LIN {X 0,Y 153.552,Z 569.709,A -85,B 0,C 180,E1 -25423.871,E2 -25423.871} C_VEL
LIN {X 0,Y 146.34,Z 578.875,A -85,B 0,C 180,E1 -25427.749,E2 -25427.749} C_VEL
LIN {X 0,Y 140.763,Z 585.487,A -85,B 0,C 180,E1 -25431.382,E2 -25431.382} C_VEL
LIN {X 0,Y 134.19,Z 592.793,A -85,B 0,C 180,E1 -25436.638,E2 -25436.638} C_VEL
LIN {X 0,Y 128.826,Z 598.573,A -85,B 0,C 180,E1 -25442.371,E2 -25442.371} C_VEL
LIN {X 0,Y 125.476,Z 601.997,A -85,B 0,C 180,E1 -25446.915,E2 -25446.915} C_VEL
LIN {X 0,Y 122.311,Z 605.447,A -85,B 0,C 180,E1 -25453.302,E2 -25453.302} C_VEL
LIN {X 0,Y 120.389,Z 607.718,A -85,B 0,C 180,E1 -25459.912,E2 -25459.912} C_VEL
LIN {X 0,Y 119.599,Z 608.867,A -85,B 0,C 180,E1 -25466.63,E2 -25466.63} C_VEL
LIN {X 0,Y 119.528,Z 608.954,A -85,B 0,C 180,E1 -25471.681,E2 -25471.681} C_VEL
LIN {X 0,Y 119.898,Z 608.461,A -85,B 0,C 180,E1 -25476.731,E2 -25476.731} C_VEL
LIN {X 0,Y 121.179,Z 606.8,A -85,B 0,C 180,E1 -25483.413,E2 -25483.413} C_VEL
LIN {X 0,Y 123.696,Z 603.988,A -85,B 0,C 180,E1 -25489.93,E2 -25489.93} C_VEL
LIN {X 0,Y 127.583,Z 599.947,A -85,B 0,C 180,E1 -25496.146,E2 -25496.146} C_VEL
LIN {X 0,Y 132.603,Z 594.585,A -85,B 0,C 180,E1 -25502.004,E2 -25502.004} C_VEL
LIN {X 0,Y 138.944,Z 587.736,A -85,B 0,C 180,E1 -25507.37,E2 -25507.37} C_VEL
LIN {X 0,Y 146.247,Z 579.18,A -85,B 0,C 180,E1 -25512.28,E2 -25512.28} C_VEL
LIN {X 0,Y 153.435,Z 570.072,A -85,B 0,C 180,E1 -25516.17,E2 -25516.17} C_VEL
LIN {X 0,Y 159.977,Z 560.798,A -85,B 0,C 180,E1 -25519.27,E2 -25519.27} C_VEL
LIN {X 0,Y 167.681,Z 548.768,A -85,B 0,C 180,E1 -25522.287,E2 -25522.287} C_VEL
LIN {X 0,Y 174.467,Z 536.481,A -85,B 0,C 180,E1 -25524.657,E2 -25524.657} C_VEL
LIN {X 0,Y 180.497,Z 523.657,A -85,B 0,C 180,E1 -25526.588,E2 -25526.588} C_VEL
LIN {X 0,Y 185.677,Z 510.287,A -85,B 0,C 180,E1 -25528.183,E2 -25528.183} C_VEL
LIN {X 0,Y 190.275,Z 495.944,A -85,B 0,C 180,E1 -25529.435,E2 -25529.435} C_VEL
LIN {X 0,Y 194.075,Z 480.371,A -85,B 0,C 180,E1 -25530.435,E2 -25530.435} C_VEL
LIN {X 0,Y 196.56,Z 465.55,A -85,B 0,C 180,E1 -25531.094,E2 -25531.094} C_VEL
LIN {X 0,Y 199.678,Z 433.456,A -85,B 0,C 180,E1 -25531.975,E2 -25531.975} C_VEL
LIN {X 0,Y 201.434,Z 413.367,A -85,B 0,C 180,E1 -25532.537,E2 -25532.537} C_VEL
LIN {X 0,Y 196.703,Z 403.519,A -85,B 0,C 180,E1 -25536.219,E2 -25536.219} C_VEL
LIN {X 0,Y 193.073,Z 396.884,A -85,B 0,C 180,E1 -25539.518,E2 -25539.518} C_VEL
LIN {X 0,Y 190.075,Z 391.565,A -85,B 0,C 180,E1 -25542.794,E2 -25542.794} C_VEL
LIN {X 0,Y 187.731,Z 387.7,A -85,B 0,C 180,E1 -25545.916,E2 -25545.916} C_VEL
LIN {X 0,Y 185.703,Z 383.97,A -85,B 0,C 180,E1 -25549.506,E2 -25549.506} C_VEL
LIN {X 0,Y 183.861,Z 381,A -85,B 0,C 180,E1 -25554.558,E2 -25554.558} C_VEL
LIN {X 0,Y 183.557,Z 379.432,A -85,B 0,C 180,E1 -25556.707,E2 -25556.707} C_VEL
LIN {X 0,Y 183.337,Z 379.121,A -85,B 0,C 180,E1 -25560,E2 -25560} C_VEL
LIN {X 0,Y 183.568,Z 379.555,A -85,B 0,C 180,E1 -25562.949,E2 -25562.949} C_VEL
LIN {X 0,Y 185.21,Z 383.47,A -85,B 0,C 180,E1 -25569.005,E2 -25569.005} C_VEL
LIN {X 0,Y 185.94,Z 384.419,A -85,B 0,C 180,E1 -25570.491,E2 -25570.491} C_VEL
LIN {X 0,Y 188.426,Z 388.76,A -85,B 0,C 180,E1 -25574.582,E2 -25574.582} C_VEL
LIN {X 0,Y 190.981,Z 393.14,A -85,B 0,C 180,E1 -25577.773,E2 -25577.773} C_VEL
LIN {X 0,Y 193.616,Z 397.814,A -85,B 0,C 180,E1 -25580.518,E2 -25580.518} C_VEL
LIN {X 0,Y 196.945,Z 405.983,A -85,B 0,C 180,E1 -25583.669,E2 -25583.669} C_VEL
LIN {X 0,Y 200.304,Z 415.239,A -85,B 0,C 180,E1 -25586.483,E2 -25586.483} C_VEL
LIN {X 0,Y 201.157,Z 417.755,A -85,B 0,C 180,E1 -25587.153,E2 -25587.153} C_VEL
LIN {X 0,Y 196.088,Z 472.023,A -85,B 0,C 180,E1 -25588.616,E2 -25588.616} C_VEL
LIN {X 0,Y 193.318,Z 487.832,A -85,B 0,C 180,E1 -25589.25,E2 -25589.25} C_VEL
LIN {X 0,Y 189.505,Z 503.063,A -85,B 0,C 180,E1 -25590.168,E2 -25590.168} C_VEL
LIN {X 0,Y 184.942,Z 516.79,A -85,B 0,C 180,E1 -25591.239,E2 -25591.239} C_VEL
LIN {X 0,Y 179.479,Z 530.244,A -85,B 0,C 180,E1 -25592.661,E2 -25592.661} C_VEL
LIN {X 0,Y 173.308,Z 543.167,A -85,B 0,C 180,E1 -25594.487,E2 -25594.487} C_VEL
LIN {X 0,Y 166.611,Z 555.308,A -85,B 0,C 180,E1 -25596.732,E2 -25596.732} C_VEL
LIN {X 0,Y 159.273,Z 566.801,A -85,B 0,C 180,E1 -25599.45,E2 -25599.45} C_VEL
LIN {X 0,Y 152.418,Z 576.486,A -85,B 0,C 180,E1 -25602.461,E2 -25602.461} C_VEL
LIN {X 0,Y 145.046,Z 586.009,A -85,B 0,C 180,E1 -25606.335,E2 -25606.335} C_VEL
LIN {X 0,Y 138.531,Z 593.959,A -85,B 0,C 180,E1 -25610.644,E2 -25610.644} C_VEL
LIN {X 0,Y 131.988,Z 601.387,A -85,B 0,C 180,E1 -25616.008,E2 -25616.008} C_VEL
LIN {X 0,Y 127.784,Z 606.137,A -85,B 0,C 180,E1 -25620.565,E2 -25620.565} C_VEL
LIN {X 0,Y 125.367,Z 608.182,A -85,B 0,C 180,E1 -25622.835,E2 -25622.835} C_VEL
LIN {X 0,Y 120.068,Z 611.099,A -85,B 0,C 180,E1 -25626.514,E2 -25626.514} C_VEL
LIN {X 0,Y 116.037,Z 613.032,A -85,B 0,C 180,E1 -25629.711,E2 -25629.711} C_VEL
LIN {X 0,Y 113.983,Z 614.267,A -85,B 0,C 180,E1 -25632.41,E2 -25632.41} C_VEL
LIN {X 0,Y 113.609,Z 614.613,A -85,B 0,C 180,E1 -25633.367,E2 -25633.367} C_VEL
LIN {X 0,Y 112.455,Z 616.484,A -85,B 0,C 180,E1 -25639.195,E2 -25639.195} C_VEL
LIN {X 0,Y 112.168,Z 617.688,A -85,B 0,C 180,E1 -25646.409,E2 -25646.409} C_VEL
LIN {X 0,Y 112.361,Z 617.854,A -85,B 0,C 180,E1 -25650.002,E2 -25650.002} C_VEL
LIN {X 0,Y 112.191,Z 617.211,A -85,B 0,C 180,E1 -25657.199,E2 -25657.199} C_VEL
LIN {X 0,Y 113.057,Z 615.402,A -85,B 0,C 180,E1 -25664.4,E2 -25664.4} C_VEL
LIN {X 0,Y 115.446,Z 612.422,A -85,B 0,C 180,E1 -25671.426,E2 -25671.426} C_VEL
LIN {X 0,Y 119.303,Z 608.201,A -85,B 0,C 180,E1 -25678.119,E2 -25678.119} C_VEL
LIN {X 0,Y 124.542,Z 602.629,A -85,B 0,C 180,E1 -25684.356,E2 -25684.356} C_VEL
LIN {X 0,Y 131.241,Z 595.569,A -85,B 0,C 180,E1 -25689.988,E2 -25689.988} C_VEL
LIN {X 0,Y 137.341,Z 588.55,A -85,B 0,C 180,E1 -25694.242,E2 -25694.242} C_VEL
LIN {X 0,Y 145.382,Z 578.944,A -85,B 0,C 180,E1 -25698.531,E2 -25698.531} C_VEL
LIN {X 0,Y 153.568,Z 568.039,A -85,B 0,C 180,E1 -25702.135,E2 -25702.135} C_VEL
LIN {X 0,Y 161.782,Z 555.793,A -85,B 0,C 180,E1 -25705.082,E2 -25705.082} C_VEL
LIN {X 0,Y 168.964,Z 543.304,A -85,B 0,C 180,E1 -25707.385,E2 -25707.385} C_VEL
LIN {X 0,Y 175.041,Z 531.032,A -85,B 0,C 180,E1 -25709.119,E2 -25709.119} C_VEL
LIN {X 0,Y 180.613,Z 517.76,A -85,B 0,C 180,E1 -25710.537,E2 -25710.537} C_VEL
LIN {X 0,Y 185.274,Z 504.367,A -85,B 0,C 180,E1 -25711.593,E2 -25711.593} C_VEL
LIN {X 0,Y 189.234,Z 489.693,A -85,B 0,C 180,E1 -25712.464,E2 -25712.464} C_VEL
LIN {X 0,Y 192.151,Z 474.204,A -85,B 0,C 180,E1 -25713.128,E2 -25713.128} C_VEL
LIN {X 0,Y 194.293,Z 455.279,A -85,B 0,C 180,E1 -25713.639,E2 -25713.639} C_VEL
LIN {X 0,Y 197.478,Z 420.453,A -85,B 0,C 180,E1 -25714.578,E2 -25714.578} C_VEL
LIN {X 0,Y 194.285,Z 411.099,A -85,B 0,C 180,E1 -25717.467,E2 -25717.467} C_VEL
LIN {X 0,Y 191.368,Z 403.557,A -85,B 0,C 180,E1 -25720.442,E2 -25720.442} C_VEL
LIN {X 0,Y 188.462,Z 398.084,A -85,B 0,C 180,E1 -25723.759,E2 -25723.759} C_VEL
LIN {X 0,Y 186.121,Z 394.028,A -85,B 0,C 180,E1 -25727.044,E2 -25727.044} C_VEL
LIN {X 0,Y 184.324,Z 390.657,A -85,B 0,C 180,E1 -25730.398,E2 -25730.398} C_VEL
LIN {X 0,Y 182.51,Z 387.017,A -85,B 0,C 180,E1 -25736.136,E2 -25736.136} C_VEL
LIN {X 0,Y 182.38,Z 386.274,A -85,B 0,C 180,E1 -25737.239,E2 -25737.239} C_VEL
LIN {X 0,Y 182.237,Z 386.167,A -85,B 0,C 180,E1 -25742.21,E2 -25742.21} C_VEL
LIN {X 0,Y 182.454,Z 386.689,A -85,B 0,C 180,E1 -25744.004,E2 -25744.004} C_VEL
LIN {X 0,Y 183.802,Z 390.149,A -85,B 0,C 180,E1 -25749.075,E2 -25749.075} C_VEL
LIN {X 0,Y 184.618,Z 391.329,A -85,B 0,C 180,E1 -25750.834,E2 -25750.834} C_VEL
LIN {X 0,Y 186.972,Z 395.589,A -85,B 0,C 180,E1 -25754.837,E2 -25754.837} C_VEL
LIN {X 0,Y 189.331,Z 399.838,A -85,B 0,C 180,E1 -25757.904,E2 -25757.904} C_VEL
LIN {X 0,Y 192.068,Z 404.893,A -85,B 0,C 180,E1 -25760.849,E2 -25760.849} C_VEL
LIN {X 0,Y 195.488,Z 411.77,A -85,B 0,C 180,E1 -25763.998,E2 -25763.998} C_VEL
LIN {X 0,Y 197.747,Z 416.775,A -85,B 0,C 180,E1 -25765.862,E2 -25765.862} C_VEL
LIN {X 0,Y 193.157,Z 465.028,A -85,B 0,C 180,E1 -25767.189,E2 -25767.189} C_VEL
LIN {X 0,Y 190.472,Z 480.44,A -85,B 0,C 180,E1 -25767.82,E2 -25767.82} C_VEL
LIN {X 0,Y 186.85,Z 495.126,A -85,B 0,C 180,E1 -25768.732,E2 -25768.732} C_VEL
LIN {X 0,Y 182.161,Z 509.686,A -85,B 0,C 180,E1 -25769.984,E2 -25769.984} C_VEL
LIN {X 0,Y 177.053,Z 522.601,A -85,B 0,C 180,E1 -25771.474,E2 -25771.474} C_VEL
LIN {X 0,Y 170.555,Z 536.147,A -85,B 0,C 180,E1 -25773.441,E2 -25773.441} C_VEL
LIN {X 0,Y 163.521,Z 548.533,A -85,B 0,C 180,E1 -25775.781,E2 -25775.781} C_VEL
LIN {X 0,Y 156.694,Z 558.904,A -85,B 0,C 180,E1 -25778.286,E2 -25778.286} C_VEL
LIN {X 0,Y 149.799,Z 568.511,A -85,B 0,C 180,E1 -25781.35,E2 -25781.35} C_VEL
LIN {X 0,Y 143.255,Z 576.708,A -85,B 0,C 180,E1 -25784.652,E2 -25784.652} C_VEL
LIN {X 0,Y 136.203,Z 584.763,A -85,B 0,C 180,E1 -25788.858,E2 -25788.858} C_VEL
LIN {X 0,Y 129.928,Z 591.404,A -85,B 0,C 180,E1 -25793.485,E2 -25793.485} C_VEL
LIN {X 0,Y 123.831,Z 597.54,A -85,B 0,C 180,E1 -25799.281,E2 -25799.281} C_VEL
LIN {X 0,Y 118.956,Z 602.269,A -85,B 0,C 180,E1 -25805.569,E2 -25805.569} C_VEL
LIN {X 0,Y 115.513,Z 605.719,A -85,B 0,C 180,E1 -25812.288,E2 -25812.288} C_VEL
LIN {X 0,Y 113.386,Z 607.989,A -85,B 0,C 180,E1 -25819.282,E2 -25819.282} C_VEL
LIN {X 0,Y 112.523,Z 609.137,A -85,B 0,C 180,E1 -25826.417,E2 -25826.417} C_VEL
LIN {X 0,Y 112.46,Z 609.266,A -85,B 0,C 180,E1 -25830.803,E2 -25830.803} C_VEL
LIN {X 0,Y 112.854,Z 608.731,A -85,B 0,C 180,E1 -25837.153,E2 -25837.153} C_VEL
LIN {X 0,Y 114.26,Z 607.071,A -85,B 0,C 180,E1 -25844.241,E2 -25844.241} C_VEL
LIN {X 0,Y 117.025,Z 604.258,A -85,B 0,C 180,E1 -25851.119,E2 -25851.119} C_VEL
LIN {X 0,Y 121.225,Z 600.217,A -85,B 0,C 180,E1 -25857.631,E2 -25857.631} C_VEL
LIN {X 0,Y 126.622,Z 594.855,A -85,B 0,C 180,E1 -25863.712,E2 -25863.712} C_VEL
LIN {X 0,Y 133.356,Z 588.005,A -85,B 0,C 180,E1 -25869.227,E2 -25869.227} C_VEL
LIN {X 0,Y 141.056,Z 579.449,A -85,B 0,C 180,E1 -25874.228,E2 -25874.228} C_VEL
LIN {X 0,Y 147.522,Z 571.748,A -85,B 0,C 180,E1 -25877.596,E2 -25877.596} C_VEL
LIN {X 0,Y 154.236,Z 562.683,A -85,B 0,C 180,E1 -25880.77,E2 -25880.77} C_VEL
LIN {X 0,Y 161.56,Z 551.969,A -85,B 0,C 180,E1 -25883.586,E2 -25883.586} C_VEL
LIN {X 0,Y 168.484,Z 540.271,A -85,B 0,C 180,E1 -25886,E2 -25886} C_VEL
LIN {X 0,Y 174.929,Z 527.738,A -85,B 0,C 180,E1 -25887.974,E2 -25887.974} C_VEL
LIN {X 0,Y 180.224,Z 515.305,A -85,B 0,C 180,E1 -25889.573,E2 -25889.573} C_VEL
LIN {X 0,Y 185.061,Z 501.838,A -85,B 0,C 180,E1 -25890.862,E2 -25890.862} C_VEL
LIN {X 0,Y 189.202,Z 487.184,A -85,B 0,C 180,E1 -25891.908,E2 -25891.908} C_VEL
LIN {X 0,Y 192.295,Z 471.921,A -85,B 0,C 180,E1 -25892.71,E2 -25892.71} C_VEL
LIN {X 0,Y 194.29,Z 456.851,A -85,B 0,C 180,E1 -25893.198,E2 -25893.198} C_VEL
LIN {X 0,Y 198,Z 416.982,A -85,B 0,C 180,E1 -25894.238,E2 -25894.238} C_VEL
LIN {X 0,Y 194.142,Z 408.687,A -85,B 0,C 180,E1 -25897.519,E2 -25897.519} C_VEL
LIN {X 0,Y 190.419,Z 401.503,A -85,B 0,C 180,E1 -25901.263,E2 -25901.263} C_VEL
LIN {X 0,Y 188.03,Z 397.319,A -85,B 0,C 180,E1 -25904.152,E2 -25904.152} C_VEL
LIN {X 0,Y 186.393,Z 394.382,A -85,B 0,C 180,E1 -25906.546,E2 -25906.546} C_VEL
LIN {X 0,Y 184.5,Z 390.792,A -85,B 0,C 180,E1 -25910.13,E2 -25910.13} C_VEL
LIN {X 0,Y 182.75,Z 387.32,A -85,B 0,C 180,E1 -25915.865,E2 -25915.865} C_VEL
LIN {X 0,Y 182.622,Z 386.361,A -85,B 0,C 180,E1 -25917.242,E2 -25917.242} C_VEL
LIN {X 0,Y 182.617,Z 386.338,A -85,B 0,C 180,E1 -25922.205,E2 -25922.205} C_VEL
LIN {X 0,Y 184.348,Z 390.581,A -85,B 0,C 180,E1 -25929.048,E2 -25929.048} C_VEL
LIN {X 0,Y 184.802,Z 391.299,A -85,B 0,C 180,E1 -25930.026,E2 -25930.026} C_VEL
LIN {X 0,Y 187.075,Z 395.482,A -85,B 0,C 180,E1 -25933.995,E2 -25933.995} C_VEL
LIN {X 0,Y 189.336,Z 399.547,A -85,B 0,C 180,E1 -25936.996,E2 -25936.996} C_VEL
LIN {X 0,Y 191.684,Z 403.991,A -85,B 0,C 180,E1 -25939.615,E2 -25939.615} C_VEL
LIN {X 0,Y 194.459,Z 411.21,A -85,B 0,C 180,E1 -25942.455,E2 -25942.455} C_VEL
LIN {X 0,Y 197.488,Z 420.003,A -85,B 0,C 180,E1 -25945.209,E2 -25945.209} C_VEL
LIN {X 0,Y 197.736,Z 420.842,A -85,B 0,C 180,E1 -25945.429,E2 -25945.429} C_VEL
LIN {X 0,Y 192.751,Z 471.989,A -85,B 0,C 180,E1 -25946.769,E2 -25946.769} C_VEL
LIN {X 0,Y 189.948,Z 487.57,A -85,B 0,C 180,E1 -25947.38,E2 -25947.38} C_VEL
LIN {X 0,Y 186.032,Z 502.8,A -85,B 0,C 180,E1 -25948.274,E2 -25948.274} C_VEL
LIN {X 0,Y 181.359,Z 516.525,A -85,B 0,C 180,E1 -25949.32,E2 -25949.32} C_VEL
LIN {X 0,Y 175.741,Z 529.978,A -85,B 0,C 180,E1 -25950.708,E2 -25950.708} C_VEL
LIN {X 0,Y 168.962,Z 543.687,A -85,B 0,C 180,E1 -25952.618,E2 -25952.618} C_VEL
LIN {X 0,Y 161.8,Z 556.113,A -85,B 0,C 180,E1 -25954.931,E2 -25954.931} C_VEL
LIN {X 0,Y 153.607,Z 568.295,A -85,B 0,C 180,E1 -25957.887,E2 -25957.887} C_VEL
LIN {X 0,Y 145.38,Z 579.146,A -85,B 0,C 180,E1 -25961.472,E2 -25961.472} C_VEL
LIN {X 0,Y 137.695,Z 588.394,A -85,B 0,C 180,E1 -25965.607,E2 -25965.607} C_VEL
LIN {X 0,Y 131.243,Z 595.726,A -85,B 0,C 180,E1 -25970.016,E2 -25970.016} C_VEL
LIN {X 0,Y 124.559,Z 602.748,A -85,B 0,C 180,E1 -25975.653,E2 -25975.653} C_VEL
LIN {X 0,Y 118.779,Z 608.82,A -85,B 0,C 180,E1 -25982.564,E2 -25982.564} C_VEL
LIN {X 0,Y 115.444,Z 612.489,A -85,B 0,C 180,E1 -25988.578,E2 -25988.578} C_VEL
LIN {X 0,Y 113.609,Z 614.613,A -85,B 0,C 180,E1 -25993.367,E2 -25993.367} C_VEL
LIN {X 0,Y 112.237,Z 615.668,A -85,B 0,C 180,E1 -25996.238,E2 -25996.238} C_VEL
LIN {X 0,Y 108.69,Z 616.831,A -85,B 0,C 180,E1 -26001.006,E2 -26001.006} C_VEL
LIN {X 0,Y 106.114,Z 617.35,A -85,B 0,C 180,E1 -26005.038,E2 -26005.038} C_VEL
LIN {X 0,Y 105.198,Z 617.515,A -85,B 0,C 180,E1 -26008.232,E2 -26008.232} C_VEL
LIN {X 0,Y 105.202,Z 617.554,A -85,B 0,C 180,E1 -26009.314,E2 -26009.314} C_VEL
LIN {X 0,Y 105.081,Z 617.411,A -85,B 0,C 180,E1 -26013.837,E2 -26013.837} C_VEL
LIN {X 0,Y 105.455,Z 616.179,A -85,B 0,C 180,E1 -26021.535,E2 -26021.535} C_VEL
LIN {X 0,Y 107.235,Z 613.787,A -85,B 0,C 180,E1 -26029.131,E2 -26029.131} C_VEL
LIN {X 0,Y 110.722,Z 610.198,A -85,B 0,C 180,E1 -26036.382,E2 -26036.382} C_VEL
LIN {X 0,Y 115.67,Z 605.317,A -85,B 0,C 180,E1 -26043.152,E2 -26043.152} C_VEL
LIN {X 0,Y 122.065,Z 599.021,A -85,B 0,C 180,E1 -26049.299,E2 -26049.299} C_VEL
LIN {X 0,Y 128.724,Z 592.235,A -85,B 0,C 180,E1 -26054.118,E2 -26054.118} C_VEL
LIN {X 0,Y 136.134,Z 584.034,A -85,B 0,C 180,E1 -26058.469,E2 -26058.469} C_VEL
LIN {X 0,Y 144.342,Z 574.22,A -85,B 0,C 180,E1 -26062.301,E2 -26062.301} C_VEL
LIN {X 0,Y 151.875,Z 564.194,A -85,B 0,C 180,E1 -26065.226,E2 -26065.226} C_VEL
LIN {X 0,Y 159.467,Z 552.848,A -85,B 0,C 180,E1 -26067.734,E2 -26067.734} C_VEL
LIN {X 0,Y 166.593,Z 540.433,A -85,B 0,C 180,E1 -26069.865,E2 -26069.865} C_VEL
LIN {X 0,Y 172.931,Z 527.625,A -85,B 0,C 180,E1 -26071.507,E2 -26071.507} C_VEL
LIN {X 0,Y 178.678,Z 513.643,A -85,B 0,C 180,E1 -26072.865,E2 -26072.865} C_VEL
LIN {X 0,Y 183.496,Z 499.24,A -85,B 0,C 180,E1 -26073.856,E2 -26073.856} C_VEL
LIN {X 0,Y 187.171,Z 484.445,A -85,B 0,C 180,E1 -26074.63,E2 -26074.63} C_VEL
LIN {X 0,Y 189.572,Z 470.621,A -85,B 0,C 180,E1 -26075.143,E2 -26075.143} C_VEL
LIN {X 0,Y 194.235,Z 423.709,A -85,B 0,C 180,E1 -26076.35,E2 -26076.35} C_VEL
LIN {X 0,Y 191.745,Z 415.955,A -85,B 0,C 180,E1 -26078.851,E2 -26078.851} C_VEL
LIN {X 0,Y 189.449,Z 409.614,A -85,B 0,C 180,E1 -26081.41,E2 -26081.41} C_VEL
LIN {X 0,Y 186.753,Z 404.322,A -85,B 0,C 180,E1 -26084.727,E2 -26084.727} C_VEL
LIN {X 0,Y 184.823,Z 400.755,A -85,B 0,C 180,E1 -26087.65,E2 -26087.65} C_VEL
LIN {X 0,Y 183.263,Z 397.581,A -85,B 0,C 180,E1 -26090.759,E2 -26090.759} C_VEL
LIN {X 0,Y 181.61,Z 394.108,A -85,B 0,C 180,E1 -26096.256,E2 -26096.256} C_VEL
LIN {X 0,Y 181.442,Z 393.23,A -85,B 0,C 180,E1 -26097.78,E2 -26097.78} C_VEL
LIN {X 0,Y 181.43,Z 393.295,A -85,B 0,C 180,E1 -26102.776,E2 -26102.776} C_VEL
LIN {X 0,Y 181.639,Z 394.346,A -85,B 0,C 180,E1 -26104.577,E2 -26104.577} C_VEL
LIN {X 0,Y 183.057,Z 397.424,A -85,B 0,C 180,E1 -26109.391,E2 -26109.391} C_VEL
LIN {X 0,Y 183.734,Z 398.826,A -85,B 0,C 180,E1 -26110.922,E2 -26110.922} C_VEL
LIN {X 0,Y 185.722,Z 402.449,A -85,B 0,C 180,E1 -26114.379,E2 -26114.379} C_VEL
LIN {X 0,Y 188.542,Z 407.745,A -85,B 0,C 180,E1 -26118.122,E2 -26118.122} C_VEL
LIN {X 0,Y 191.93,Z 414.739,A -85,B 0,C 180,E1 -26121.748,E2 -26121.748} C_VEL
LIN {X 0,Y 194.481,Z 420.422,A -85,B 0,C 180,E1 -26124.101,E2 -26124.101} C_VEL
LIN {X 0,Y 190.029,Z 465.302,A -85,B 0,C 180,E1 -26125.291,E2 -26125.291} C_VEL
LIN {X 0,Y 187.451,Z 479.864,A -85,B 0,C 180,E1 -26125.863,E2 -26125.863} C_VEL
LIN {X 0,Y 183.541,Z 495.404,A -85,B 0,C 180,E1 -26126.788,E2 -26126.788} C_VEL
LIN {X 0,Y 178.728,Z 509.962,A -85,B 0,C 180,E1 -26128.017,E2 -26128.017} C_VEL
LIN {X 0,Y 173.336,Z 523.154,A -85,B 0,C 180,E1 -26129.51,E2 -26129.51} C_VEL
LIN {X 0,Y 166.76,Z 536.421,A -85,B 0,C 180,E1 -26131.411,E2 -26131.411} C_VEL
LIN {X 0,Y 159.474,Z 548.807,A -85,B 0,C 180,E1 -26133.712,E2 -26133.712} C_VEL
LIN {X 0,Y 152.396,Z 559.178,A -85,B 0,C 180,E1 -26136.189,E2 -26136.189} C_VEL
LIN {X 0,Y 145.179,Z 568.785,A -85,B 0,C 180,E1 -26139.234,E2 -26139.234} C_VEL
LIN {X 0,Y 138.352,Z 576.981,A -85,B 0,C 180,E1 -26142.558,E2 -26142.558} C_VEL
LIN {X 0,Y 130.922,Z 585.036,A -85,B 0,C 180,E1 -26146.807,E2 -26146.807} C_VEL
LIN {X 0,Y 124.262,Z 591.678,A -85,B 0,C 180,E1 -26151.525,E2 -26151.525} C_VEL
LIN {X 0,Y 117.751,Z 597.814,A -85,B 0,C 180,E1 -26157.507,E2 -26157.507} C_VEL
LIN {X 0,Y 112.515,Z 602.541,A -85,B 0,C 180,E1 -26164.07,E2 -26164.07} C_VEL
LIN {X 0,Y 108.762,Z 605.99,A -85,B 0,C 180,E1 -26171.148,E2 -26171.148} C_VEL
LIN {X 0,Y 106.409,Z 608.261,A -85,B 0,C 180,E1 -26178.57,E2 -26178.57} C_VEL
LIN {X 0,Y 105.455,Z 609.407,A -85,B 0,C 180,E1 -26186.177,E2 -26186.177} C_VEL
LIN {X 0,Y 105.392,Z 609.558,A -85,B 0,C 180,E1 -26189.998,E2 -26189.998} C_VEL
LIN {X 0,Y 105.807,Z 609.001,A -85,B 0,C 180,E1 -26197.632,E2 -26197.632} C_VEL
LIN {X 0,Y 107.38,Z 607.342,A -85,B 0,C 180,E1 -26205.175,E2 -26205.175} C_VEL
LIN {X 0,Y 110.393,Z 604.529,A -85,B 0,C 180,E1 -26212.455,E2 -26212.455} C_VEL
LIN {X 0,Y 114.961,Z 600.488,A -85,B 0,C 180,E1 -26219.278,E2 -26219.278} C_VEL
LIN {X 0,Y 120.749,Z 595.126,A -85,B 0,C 180,E1 -26225.592,E2 -26225.592} C_VEL
LIN {X 0,Y 127.898,Z 588.276,A -85,B 0,C 180,E1 -26231.252,E2 -26231.252} C_VEL
LIN {X 0,Y 136.043,Z 579.719,A -85,B 0,C 180,E1 -26236.321,E2 -26236.321} C_VEL
LIN {X 0,Y 142.807,Z 572.017,A -85,B 0,C 180,E1 -26239.71,E2 -26239.71} C_VEL
LIN {X 0,Y 149.839,Z 562.951,A -85,B 0,C 180,E1 -26242.877,E2 -26242.877} C_VEL
LIN {X 0,Y 157.449,Z 552.236,A -85,B 0,C 180,E1 -26245.665,E2 -26245.665} C_VEL
LIN {X 0,Y 164.623,Z 540.537,A -85,B 0,C 180,E1 -26248.046,E2 -26248.046} C_VEL
LIN {X 0,Y 171.771,Z 526.96,A -85,B 0,C 180,E1 -26250.13,E2 -26250.13} C_VEL
LIN {X 0,Y 177.492,Z 513.632,A -85,B 0,C 180,E1 -26251.763,E2 -26251.763} C_VEL
LIN {X 0,Y 182.758,Z 498.723,A -85,B 0,C 180,E1 -26253.083,E2 -26253.083} C_VEL
LIN {X 0,Y 186.857,Z 483.643,A -85,B 0,C 180,E1 -26254.045,E2 -26254.045} C_VEL
LIN {X 0,Y 189.664,Z 468.983,A -85,B 0,C 180,E1 -26254.725,E2 -26254.725} C_VEL
LIN {X 0,Y 191.551,Z 453.831,A -85,B 0,C 180,E1 -26255.153,E2 -26255.153} C_VEL
LIN {X 0,Y 194.707,Z 420.604,A -85,B 0,C 180,E1 -26256.023,E2 -26256.023} C_VEL
LIN {X 0,Y 191.485,Z 413.416,A -85,B 0,C 180,E1 -26259.056,E2 -26259.056} C_VEL
LIN {X 0,Y 188.157,Z 406.822,A -85,B 0,C 180,E1 -26262.753,E2 -26262.753} C_VEL
LIN {X 0,Y 186.031,Z 402.882,A -85,B 0,C 180,E1 -26265.645,E2 -26265.645} C_VEL
LIN {X 0,Y 184.963,Z 400.87,A -85,B 0,C 180,E1 -26267.38,E2 -26267.38} C_VEL
LIN {X 0,Y 183.383,Z 397.654,A -85,B 0,C 180,E1 -26270.626,E2 -26270.626} C_VEL
LIN {X 0,Y 181.802,Z 394.148,A -85,B 0,C 180,E1 -26276.398,E2 -26276.398} C_VEL
LIN {X 0,Y 181.701,Z 393.312,A -85,B 0,C 180,E1 -26277.783,E2 -26277.783} C_VEL
LIN {X 0,Y 181.743,Z 393.458,A -85,B 0,C 180,E1 -26282.216,E2 -26282.216} C_VEL
LIN {X 0,Y 183.238,Z 397.453,A -85,B 0,C 180,E1 -26288.547,E2 -26288.547} C_VEL
LIN {X 0,Y 183.771,Z 398.434,A -85,B 0,C 180,E1 -26289.782,E2 -26289.782} C_VEL
LIN {X 0,Y 185.745,Z 402.2,A -85,B 0,C 180,E1 -26293.4,E2 -26293.4} C_VEL
LIN {X 0,Y 188.113,Z 406.656,A -85,B 0,C 180,E1 -26296.691,E2 -26296.691} C_VEL
LIN {X 0,Y 190.081,Z 410.84,A -85,B 0,C 180,E1 -26299.016,E2 -26299.016} C_VEL
LIN {X 0,Y 192.584,Z 418.01,A -85,B 0,C 180,E1 -26301.754,E2 -26301.754} C_VEL
LIN {X 0,Y 194.489,Z 423.973,A -85,B 0,C 180,E1 -26303.643,E2 -26303.643} C_VEL
LIN {X 0,Y 189.624,Z 471.934,A -85,B 0,C 180,E1 -26304.858,E2 -26304.858} C_VEL
LIN {X 0,Y 186.789,Z 487.309,A -85,B 0,C 180,E1 -26305.446,E2 -26305.446} C_VEL
LIN {X 0,Y 182.775,Z 502.536,A -85,B 0,C 180,E1 -26306.313,E2 -26306.313} C_VEL
LIN {X 0,Y 177.979,Z 516.26,A -85,B 0,C 180,E1 -26307.32,E2 -26307.32} C_VEL
LIN {X 0,Y 172.212,Z 529.711,A -85,B 0,C 180,E1 -26308.669,E2 -26308.669} C_VEL
LIN {X 0,Y 165.233,Z 543.42,A -85,B 0,C 180,E1 -26310.538,E2 -26310.538} C_VEL
LIN {X 0,Y 157.821,Z 555.845,A -85,B 0,C 180,E1 -26312.806,E2 -26312.806} C_VEL
LIN {X 0,Y 149.325,Z 568.026,A -85,B 0,C 180,E1 -26315.723,E2 -26315.723} C_VEL
LIN {X 0,Y 140.739,Z 578.875,A -85,B 0,C 180,E1 -26319.286,E2 -26319.286} C_VEL
LIN {X 0,Y 133.934,Z 586.709,A -85,B 0,C 180,E1 -26322.726,E2 -26322.726} C_VEL
LIN {X 0,Y 125.829,Z 595.454,A -85,B 0,C 180,E1 -26327.916,E2 -26327.916} C_VEL
LIN {X 0,Y 118.7,Z 602.476,A -85,B 0,C 180,E1 -26333.697,E2 -26333.697} C_VEL
LIN {X 0,Y 112.979,Z 608.014,A -85,B 0,C 180,E1 -26340.157,E2 -26340.157} C_VEL
LIN {X 0,Y 108.787,Z 612.216,A -85,B 0,C 180,E1 -26347.195,E2 -26347.195} C_VEL
LIN {X 0,Y 106.14,Z 615.176,A -85,B 0,C 180,E1 -26354.643,E2 -26354.643} C_VEL
LIN {X 0,Y 105.119,Z 616.959,A -85,B 0,C 180,E1 -26362.318,E2 -26362.318} C_VEL
LIN {X 0,Y 105.202,Z 617.554,A -85,B 0,C 180,E1 -26369.314,E2 -26369.314} C_VEL
LIN {X 0,Y 105.014,Z 617.581,A -85,B 0,C 180,E1 -26371.442,E2 -26371.442} C_VEL
LIN {X 0,Y 103.723,Z 617.402,A -85,B 0,C 180,E1 -26374.605,E2 -26374.605} C_VEL
LIN {X 0,Y 99.655,Z 616.073,A -85,B 0,C 180,E1 -26382.167,E2 -26382.167} C_VEL
LIN {X 0,Y 99.123,Z 615.13,A -85,B 0,C 180,E1 -26385.587,E2 -26385.587} C_VEL
LIN {X 0,Y 99.307,Z 614.768,A -85,B 0,C 180,E1 -26386.723,E2 -26386.723} C_VEL
LIN {X 0,Y 102.205,Z 611.873,A -85,B 0,C 180,E1 -26394.369,E2 -26394.369} C_VEL
LIN {X 0,Y 106.825,Z 607.651,A -85,B 0,C 180,E1 -26401.759,E2 -26401.759} C_VEL
LIN {X 0,Y 112.978,Z 602.08,A -85,B 0,C 180,E1 -26408.469,E2 -26408.469} C_VEL
LIN {X 0,Y 120.601,Z 595.02,A -85,B 0,C 180,E1 -26414.373,E2 -26414.373} C_VEL
LIN {X 0,Y 128.146,Z 587.334,A -85,B 0,C 180,E1 -26419.089,E2 -26419.089} C_VEL
LIN {X 0,Y 136.315,Z 578.393,A -85,B 0,C 180,E1 -26423.05,E2 -26423.05} C_VEL
LIN {X 0,Y 145.233,Z 567.49,A -85,B 0,C 180,E1 -26426.592,E2 -26426.592} C_VEL
LIN {X 0,Y 154.053,Z 555.242,A -85,B 0,C 180,E1 -26429.442,E2 -26429.442} C_VEL
LIN {X 0,Y 161.721,Z 542.752,A -85,B 0,C 180,E1 -26431.647,E2 -26431.647} C_VEL
LIN {X 0,Y 168.18,Z 530.48,A -85,B 0,C 180,E1 -26433.285,E2 -26433.285} C_VEL
LIN {X 0,Y 174.048,Z 517.206,A -85,B 0,C 180,E1 -26434.624,E2 -26434.624} C_VEL
LIN {X 0,Y 179.342,Z 502.683,A -85,B 0,C 180,E1 -26435.663,E2 -26435.663} C_VEL
LIN {X 0,Y 183.483,Z 487.607,A -85,B 0,C 180,E1 -26436.478,E2 -26436.478} C_VEL
LIN {X 0,Y 186.382,Z 472.363,A -85,B 0,C 180,E1 -26437.064,E2 -26437.064} C_VEL
LIN {X 0,Y 189.938,Z 439.628,A -85,B 0,C 180,E1 -26437.862,E2 -26437.862} C_VEL
LIN {X 0,Y 191.119,Z 426.649,A -85,B 0,C 180,E1 -26438.26,E2 -26438.26} C_VEL
LIN {X 0,Y 188.829,Z 419.293,A -85,B 0,C 180,E1 -26440.853,E2 -26440.853} C_VEL
LIN {X 0,Y 187.251,Z 414.935,A -85,B 0,C 180,E1 -26442.809,E2 -26442.809} C_VEL
LIN {X 0,Y 184.969,Z 410.31,A -85,B 0,C 180,E1 -26445.906,E2 -26445.906} C_VEL
LIN {X 0,Y 183.474,Z 407.325,A -85,B 0,C 180,E1 -26448.399,E2 -26448.399} C_VEL
LIN {X 0,Y 182.089,Z 404.363,A -85,B 0,C 180,E1 -26451.399,E2 -26451.399} C_VEL
LIN {X 0,Y 180.646,Z 400.826,A -85,B 0,C 180,E1 -26456.926,E2 -26456.926} C_VEL
LIN {X 0,Y 180.572,Z 400.32,A -85,B 0,C 180,E1 -26457.77,E2 -26457.77} C_VEL
LIN {X 0,Y 180.508,Z 400.258,A -85,B 0,C 180,E1 -26462.232,E2 -26462.232} C_VEL
LIN {X 0,Y 180.644,Z 400.903,A -85,B 0,C 180,E1 -26463.695,E2 -26463.695} C_VEL
LIN {X 0,Y 181.955,Z 404.282,A -85,B 0,C 180,E1 -26468.888,E2 -26468.888} C_VEL
LIN {X 0,Y 182.501,Z 405.472,A -85,B 0,C 180,E1 -26470.225,E2 -26470.225} C_VEL
LIN {X 0,Y 184.314,Z 409.02,A -85,B 0,C 180,E1 -26473.647,E2 -26473.647} C_VEL
LIN {X 0,Y 186.385,Z 413.192,A -85,B 0,C 180,E1 -26476.674,E2 -26476.674} C_VEL
LIN {X 0,Y 189.381,Z 419.498,A -85,B 0,C 180,E1 -26480.218,E2 -26480.218} C_VEL
LIN {X 0,Y 191.351,Z 424.086,A -85,B 0,C 180,E1 -26482.242,E2 -26482.242} C_VEL
LIN {X 0,Y 187.055,Z 465.958,A -85,B 0,C 180,E1 -26483.342,E2 -26483.342} C_VEL
LIN {X 0,Y 184.282,Z 481.001,A -85,B 0,C 180,E1 -26483.919,E2 -26483.919} C_VEL
LIN {X 0,Y 180.455,Z 495.683,A -85,B 0,C 180,E1 -26484.776,E2 -26484.776} C_VEL
LIN {X 0,Y 175.509,Z 510.238,A -85,B 0,C 180,E1 -26485.973,E2 -26485.973} C_VEL
LIN {X 0,Y 169.823,Z 523.719,A -85,B 0,C 180,E1 -26487.461,E2 -26487.461} C_VEL
LIN {X 0,Y 163.184,Z 536.695,A -85,B 0,C 180,E1 -26489.291,E2 -26489.291} C_VEL
LIN {X 0,Y 155.635,Z 549.082,A -85,B 0,C 180,E1 -26491.531,E2 -26491.531} C_VEL
LIN {X 0,Y 148.306,Z 559.452,A -85,B 0,C 180,E1 -26493.971,E2 -26493.971} C_VEL
LIN {X 0,Y 140.784,Z 569.059,A -85,B 0,C 180,E1 -26496.989,E2 -26496.989} C_VEL
LIN {X 0,Y 133.654,Z 577.253,A -85,B 0,C 180,E1 -26500.316,E2 -26500.316} C_VEL
LIN {X 0,Y 125.833,Z 585.309,A -85,B 0,C 180,E1 -26504.591,E2 -26504.591} C_VEL
LIN {X 0,Y 118.763,Z 591.951,A -85,B 0,C 180,E1 -26509.385,E2 -26509.385} C_VEL
LIN {X 0,Y 111.803,Z 598.086,A -85,B 0,C 180,E1 -26515.544,E2 -26515.544} C_VEL
LIN {X 0,Y 106.165,Z 602.813,A -85,B 0,C 180,E1 -26522.392,E2 -26522.392} C_VEL
LIN {X 0,Y 102.048,Z 606.262,A -85,B 0,C 180,E1 -26529.856,E2 -26529.856} C_VEL
LIN {X 0,Y 99.466,Z 608.531,A -85,B 0,C 180,E1 -26537.76,E2 -26537.76} C_VEL
LIN {X 0,Y 98.391,Z 609.677,A -85,B 0,C 180,E1 -26545.902,E2 -26545.902} C_VEL
LIN {X 0,Y 98.311,Z 609.828,A -85,B 0,C 180,E1 -26549.998,E2 -26549.998} C_VEL
LIN {X 0,Y 98.768,Z 609.272,A -85,B 0,C 180,E1 -26558.18,E2 -26558.18} C_VEL
LIN {X 0,Y 100.544,Z 607.612,A -85,B 0,C 180,E1 -26566.234,E2 -26566.234} C_VEL
LIN {X 0,Y 103.831,Z 604.801,A -85,B 0,C 180,E1 -26573.96,E2 -26573.96} C_VEL
LIN {X 0,Y 108.805,Z 600.758,A -85,B 0,C 180,E1 -26581.112,E2 -26581.112} C_VEL
LIN {X 0,Y 115.04,Z 595.396,A -85,B 0,C 180,E1 -26587.654,E2 -26587.654} C_VEL
LIN {X 0,Y 122.629,Z 588.546,A -85,B 0,C 180,E1 -26593.449,E2 -26593.449} C_VEL
LIN {X 0,Y 130.115,Z 581.179,A -85,B 0,C 180,E1 -26597.959,E2 -26597.959} C_VEL
LIN {X 0,Y 137.089,Z 573.684,A -85,B 0,C 180,E1 -26601.375,E2 -26601.375} C_VEL
LIN {X 0,Y 144.265,Z 564.997,A -85,B 0,C 180,E1 -26604.563,E2 -26604.563} C_VEL
LIN {X 0,Y 152.232,Z 554.444,A -85,B 0,C 180,E1 -26607.407,E2 -26607.407} C_VEL
LIN {X 0,Y 159.618,Z 543.138,A -85,B 0,C 180,E1 -26609.777,E2 -26609.777} C_VEL
LIN {X 0,Y 166.561,Z 530.844,A -85,B 0,C 180,E1 -26611.739,E2 -26611.739} C_VEL
LIN {X 0,Y 172.839,Z 517.398,A -85,B 0,C 180,E1 -26613.451,E2 -26613.451} C_VEL
LIN {X 0,Y 178.232,Z 503.443,A -85,B 0,C 180,E1 -26614.749,E2 -26614.749} C_VEL
LIN {X 0,Y 182.584,Z 489.092,A -85,B 0,C 180,E1 -26615.75,E2 -26615.75} C_VEL
LIN {X 0,Y 186.001,Z 473.73,A -85,B 0,C 180,E1 -26616.528,E2 -26616.528} C_VEL
LIN {X 0,Y 188.265,Z 457.913,A -85,B 0,C 180,E1 -26617.036,E2 -26617.036} C_VEL
LIN {X 0,Y 191.579,Z 424.301,A -85,B 0,C 180,E1 -26617.882,E2 -26617.882} C_VEL
LIN {X 0,Y 188.992,Z 418.377,A -85,B 0,C 180,E1 -26620.588,E2 -26620.588} C_VEL
LIN {X 0,Y 186.53,Z 413.2,A -85,B 0,C 180,E1 -26623.585,E2 -26623.585} C_VEL
LIN {X 0,Y 184.089,Z 408.166,A -85,B 0,C 180,E1 -26627.319,E2 -26627.319} C_VEL
LIN {X 0,Y 182.279,Z 404.521,A -85,B 0,C 180,E1 -26631.128,E2 -26631.128} C_VEL
LIN {X 0,Y 180.865,Z 400.85,A -85,B 0,C 180,E1 -26637.076,E2 -26637.076} C_VEL
LIN {X 0,Y 180.835,Z 400.372,A -85,B 0,C 180,E1 -26637.772,E2 -26637.772} C_VEL
LIN {X 0,Y 180.844,Z 400.495,A -85,B 0,C 180,E1 -26641.948,E2 -26641.948} C_VEL
LIN {X 0,Y 182.256,Z 404.445,A -85,B 0,C 180,E1 -26648.314,E2 -26648.314} C_VEL
LIN {X 0,Y 184.359,Z 408.728,A -85,B 0,C 180,E1 -26652.662,E2 -26652.662} C_VEL
LIN {X 0,Y 186.57,Z 413.165,A -85,B 0,C 180,E1 -26655.961,E2 -26655.961} C_VEL
LIN {X 0,Y 188.357,Z 417.301,A -85,B 0,C 180,E1 -26658.231,E2 -26658.231} C_VEL
LIN {X 0,Y 190.989,Z 425.557,A -85,B 0,C 180,E1 -26661.308,E2 -26661.308} C_VEL
LIN {X 0,Y 191.427,Z 427.043,A -85,B 0,C 180,E1 -26661.783,E2 -26661.783} C_VEL
LIN {X 0,Y 186.731,Z 471.79,A -85,B 0,C 180,E1 -26662.884,E2 -26662.884} C_VEL
LIN {X 0,Y 183.851,Z 487.049,A -85,B 0,C 180,E1 -26663.448,E2 -26663.448} C_VEL
LIN {X 0,Y 179.74,Z 502.273,A -85,B 0,C 180,E1 -26664.283,E2 -26664.283} C_VEL
LIN {X 0,Y 174.823,Z 515.994,A -85,B 0,C 180,E1 -26665.244,E2 -26665.244} C_VEL
LIN {X 0,Y 168.921,Z 529.446,A -85,B 0,C 180,E1 -26666.556,E2 -26666.556} C_VEL
LIN {X 0,Y 161.722,Z 543.152,A -85,B 0,C 180,E1 -26668.359,E2 -26668.359} C_VEL
LIN {X 0,Y 154.065,Z 555.576,A -85,B 0,C 180,E1 -26670.571,E2 -26670.571} C_VEL
LIN {X 0,Y 145.26,Z 567.755,A -85,B 0,C 180,E1 -26673.429,E2 -26673.429} C_VEL
LIN {X 0,Y 136.313,Z 578.604,A -85,B 0,C 180,E1 -26676.953,E2 -26676.953} C_VEL
LIN {X 0,Y 129.185,Z 586.438,A -85,B 0,C 180,E1 -26680.394,E2 -26680.394} C_VEL
LIN {X 0,Y 120.594,Z 595.182,A -85,B 0,C 180,E1 -26685.628,E2 -26685.628} C_VEL
LIN {X 0,Y 113.001,Z 602.204,A -85,B 0,C 180,E1 -26691.544,E2 -26691.544} C_VEL
LIN {X 0,Y 106.811,Z 607.741,A -85,B 0,C 180,E1 -26698.24,E2 -26698.24} C_VEL
LIN {X 0,Y 102.2,Z 611.943,A -85,B 0,C 180,E1 -26705.634,E2 -26705.634} C_VEL
LIN {X 0,Y 99.239,Z 614.903,A -85,B 0,C 180,E1 -26713.546,E2 -26713.546} C_VEL
LIN {X 0,Y 98.053,Z 616.688,A -85,B 0,C 180,E1 -26721.76,E2 -26721.76} C_VEL
LIN {X 0,Y 98.188,Z 617.314,A -85,B 0,C 180,E1 -26730.002,E2 -26730.002} C_VEL
LIN {X 0,Y 98.054,Z 616.667,A -85,B 0,C 180,E1 -26738.244,E2 -26738.244} C_VEL
LIN {X 0,Y 99.307,Z 614.768,A -85,B 0,C 180,E1 -26746.723,E2 -26746.723} C_VEL
LIN {X 0,Y 99.658,Z 613.704,A -85,B 0,C 180,E1 -26750.056,E2 -26750.056} C_VEL
LIN {X 0,Y 99.137,Z 611.547,A -85,B 0,C 180,E1 -26755.638,E2 -26755.638} C_VEL
LIN {X 0,Y 99.204,Z 609.554,A -85,B 0,C 180,E1 -26760.09,E2 -26760.09} C_VEL
LIN {X 0,Y 100.363,Z 607.801,A -85,B 0,C 180,E1 -26763.267,E2 -26763.267} C_VEL
LIN {X 0,Y 101.056,Z 607.142,A -85,B 0,C 180,E1 -26764.252,E2 -26764.252} C_VEL
LIN {X 0,Y 107.445,Z 601.805,A -85,B 0,C 180,E1 -26770.854,E2 -26770.854} C_VEL
LIN {X 0,Y 115.552,Z 594.743,A -85,B 0,C 180,E1 -26776.877,E2 -26776.877} C_VEL
LIN {X 0,Y 123.41,Z 587.226,A -85,B 0,C 180,E1 -26781.51,E2 -26781.51} C_VEL
LIN {X 0,Y 132.138,Z 578.119,A -85,B 0,C 180,E1 -26785.53,E2 -26785.53} C_VEL
LIN {X 0,Y 141.432,Z 567.215,A -85,B 0,C 180,E1 -26789.005,E2 -26789.005} C_VEL
LIN {X 0,Y 149.832,Z 556.004,A -85,B 0,C 180,E1 -26791.583,E2 -26791.583} C_VEL
LIN {X 0,Y 157.73,Z 543.716,A -85,B 0,C 180,E1 -26793.732,E2 -26793.732} C_VEL
LIN {X 0,Y 165.101,Z 530.205,A -85,B 0,C 180,E1 -26795.493,E2 -26795.493} C_VEL
LIN {X 0,Y 171.121,Z 516.93,A -85,B 0,C 180,E1 -26796.776,E2 -26796.776} C_VEL
LIN {X 0,Y 176.533,Z 502.405,A -85,B 0,C 180,E1 -26797.764,E2 -26797.764} C_VEL
LIN {X 0,Y 180.768,Z 487.327,A -85,B 0,C 180,E1 -26798.541,E2 -26798.541} C_VEL
LIN {X 0,Y 183.805,Z 471.669,A -85,B 0,C 180,E1 -26799.112,E2 -26799.112} C_VEL
LIN {X 0,Y 188.12,Z 431.863,A -85,B 0,C 180,E1 -26800.068,E2 -26800.068} C_VEL
LIN {X 0,Y 188.232,Z 429.835,A -85,B 0,C 180,E1 -26800.195,E2 -26800.195} C_VEL
LIN {X 0,Y 186.089,Z 422.602,A -85,B 0,C 180,E1 -26802.981,E2 -26802.981} C_VEL
LIN {X 0,Y 184.413,Z 418.654,A -85,B 0,C 180,E1 -26805.31,E2 -26805.31} C_VEL
LIN {X 0,Y 182.297,Z 414.157,A -85,B 0,C 180,E1 -26808.886,E2 -26808.886} C_VEL
LIN {X 0,Y 180.994,Z 411.203,A -85,B 0,C 180,E1 -26811.908,E2 -26811.908} C_VEL
LIN {X 0,Y 179.714,Z 407.651,A -85,B 0,C 180,E1 -26817.476,E2 -26817.476} C_VEL
LIN {X 0,Y 179.558,Z 407.173,A -85,B 0,C 180,E1 -26820,E2 -26820} C_VEL
LIN {X 0,Y 179.696,Z 407.595,A -85,B 0,C 180,E1 -26822.943,E2 -26822.943} C_VEL
LIN {X 0,Y 180.842,Z 411.102,A -85,B 0,C 180,E1 -26828.31,E2 -26828.31} C_VEL
LIN {X 0,Y 181.389,Z 412.369,A -85,B 0,C 180,E1 -26829.76,E2 -26829.76} C_VEL
LIN {X 0,Y 183.014,Z 415.747,A -85,B 0,C 180,E1 -26833.039,E2 -26833.039} C_VEL
LIN {X 0,Y 184.814,Z 419.595,A -85,B 0,C 180,E1 -26835.862,E2 -26835.862} C_VEL
LIN {X 0,Y 187.559,Z 425.758,A -85,B 0,C 180,E1 -26839.353,E2 -26839.353} C_VEL
LIN {X 0,Y 188.391,Z 427.769,A -85,B 0,C 180,E1 -26840.293,E2 -26840.293} C_VEL
LIN {X 0,Y 184.364,Z 466.243,A -85,B 0,C 180,E1 -26841.321,E2 -26841.321} C_VEL
LIN {X 0,Y 181.529,Z 481.28,A -85,B 0,C 180,E1 -26841.877,E2 -26841.877} C_VEL
LIN {X 0,Y 177.607,Z 495.96,A -85,B 0,C 180,E1 -26842.704,E2 -26842.704} C_VEL
LIN {X 0,Y 172.523,Z 510.514,A -85,B 0,C 180,E1 -26843.857,E2 -26843.857} C_VEL
LIN {X 0,Y 166.525,Z 524.311,A -85,B 0,C 180,E1 -26845.335,E2 -26845.335} C_VEL
LIN {X 0,Y 159.103,Z 538.206,A -85,B 0,C 180,E1 -26847.253,E2 -26847.253} C_VEL
LIN {X 0,Y 151.35,Z 550.388,A -85,B 0,C 180,E1 -26849.461,E2 -26849.461} C_VEL
LIN {X 0,Y 143.116,Z 561.487,A -85,B 0,C 180,E1 -26852.1,E2 -26852.1} C_VEL
LIN {X 0,Y 134.106,Z 572.244,A -85,B 0,C 180,E1 -26855.676,E2 -26855.676} C_VEL
LIN {X 0,Y 125.537,Z 581.179,A -85,B 0,C 180,E1 -26859.664,E2 -26859.664} C_VEL
LIN {X 0,Y 117.633,Z 588.574,A -85,B 0,C 180,E1 -26864.195,E2 -26864.195} C_VEL
LIN {X 0,Y 109.576,Z 595.477,A -85,B 0,C 180,E1 -26870.102,E2 -26870.102} C_VEL
LIN {X 0,Y 102.841,Z 600.886,A -85,B 0,C 180,E1 -26876.856,E2 -26876.856} C_VEL
LIN {X 0,Y 97.402,Z 604.964,A -85,B 0,C 180,E1 -26884.344,E2 -26884.344} C_VEL
LIN {X 0,Y 93.735,Z 607.812,A -85,B 0,C 180,E1 -26892.546,E2 -26892.546} C_VEL
LIN {X 0,Y 91.736,Z 609.512,A -85,B 0,C 180,E1 -26901.184,E2 -26901.184} C_VEL
LIN {X 0,Y 91.222,Z 610.098,A -85,B 0,C 180,E1 -26909.998,E2 -26909.998} C_VEL
LIN {X 0,Y 91.734,Z 609.543,A -85,B 0,C 180,E1 -26918.812,E2 -26918.812} C_VEL
LIN {X 0,Y 93.72,Z 607.883,A -85,B 0,C 180,E1 -26927.453,E2 -26927.453} C_VEL
LIN {X 0,Y 97.353,Z 605.072,A -85,B 0,C 180,E1 -26935.665,E2 -26935.665} C_VEL
LIN {X 0,Y 102.771,Z 601.029,A -85,B 0,C 180,E1 -26943.165,E2 -26943.165} C_VEL
LIN {X 0,Y 109.49,Z 595.666,A -85,B 0,C 180,E1 -26949.93,E2 -26949.93} C_VEL
LIN {X 0,Y 117.567,Z 588.815,A -85,B 0,C 180,E1 -26955.833,E2 -26955.833} C_VEL
LIN {X 0,Y 126.628,Z 580.257,A -85,B 0,C 180,E1 -26960.986,E2 -26960.986} C_VEL
LIN {X 0,Y 133.7,Z 572.895,A -85,B 0,C 180,E1 -26964.236,E2 -26964.236} C_VEL
LIN {X 0,Y 141.711,Z 563.488,A -85,B 0,C 180,E1 -26967.467,E2 -26967.467} C_VEL
LIN {X 0,Y 149.902,Z 552.77,A -85,B 0,C 180,E1 -26970.15,E2 -26970.15} C_VEL
LIN {X 0,Y 157.564,Z 541.071,A -85,B 0,C 180,E1 -26972.435,E2 -26972.435} C_VEL
LIN {X 0,Y 164.032,Z 529.699,A -85,B 0,C 180,E1 -26974.123,E2 -26974.123} C_VEL
LIN {X 0,Y 169.783,Z 517.663,A -85,B 0,C 180,E1 -26975.595,E2 -26975.595} C_VEL
LIN {X 0,Y 175.327,Z 503.706,A -85,B 0,C 180,E1 -26976.843,E2 -26976.843} C_VEL
LIN {X 0,Y 179.793,Z 489.353,A -85,B 0,C 180,E1 -26977.806,E2 -26977.806} C_VEL
LIN {X 0,Y 183.344,Z 473.741,A -85,B 0,C 180,E1 -26978.571,E2 -26978.571} C_VEL
LIN {X 0,Y 185.6,Z 458.292,A -85,B 0,C 180,E1 -26979.047,E2 -26979.047} C_VEL
LIN {X 0,Y 188.669,Z 428.045,A -85,B 0,C 180,E1 -26979.788,E2 -26979.788} C_VEL
LIN {X 0,Y 185.857,Z 421.552,A -85,B 0,C 180,E1 -26983.171,E2 -26983.171} C_VEL
LIN {X 0,Y 183.701,Z 416.938,A -85,B 0,C 180,E1 -26986.345,E2 -26986.345} C_VEL
LIN {X 0,Y 182.456,Z 414.283,A -85,B 0,C 180,E1 -26988.614,E2 -26988.614} C_VEL
LIN {X 0,Y 181.111,Z 411.278,A -85,B 0,C 180,E1 -26991.843,E2 -26991.843} C_VEL
LIN {X 0,Y 179.922,Z 407.386,A -85,B 0,C 180,E1 -26998.321,E2 -26998.321} C_VEL
LIN {X 0,Y 179.952,Z 407.501,A -85,B 0,C 180,E1 -27001.678,E2 -27001.678} C_VEL
LIN {X 0,Y 181.425,Z 411.833,A -85,B 0,C 180,E1 -27008.493,E2 -27008.493} C_VEL
LIN {X 0,Y 183.222,Z 415.79,A -85,B 0,C 180,E1 -27012.319,E2 -27012.319} C_VEL
LIN {X 0,Y 185.139,Z 419.874,A -85,B 0,C 180,E1 -27015.339,E2 -27015.339} C_VEL
LIN {X 0,Y 186.487,Z 423.268,A -85,B 0,C 180,E1 -27017.193,E2 -27017.193} C_VEL
LIN {X 0,Y 188.528,Z 430.26,A -85,B 0,C 180,E1 -27019.845,E2 -27019.845} C_VEL
LIN {X 0,Y 184.045,Z 471.793,A -85,B 0,C 180,E1 -27020.858,E2 -27020.858} C_VEL
LIN {X 0,Y 181.145,Z 486.788,A -85,B 0,C 180,E1 -27021.389,E2 -27021.389} C_VEL
LIN {X 0,Y 176.939,Z 502.009,A -85,B 0,C 180,E1 -27022.187,E2 -27022.187} C_VEL
LIN {X 0,Y 171.913,Z 515.729,A -85,B 0,C 180,E1 -27023.102,E2 -27023.102} C_VEL
LIN {X 0,Y 165.868,Z 529.18,A -85,B 0,C 180,E1 -27024.361,E2 -27024.361} C_VEL
LIN {X 0,Y 158.454,Z 542.884,A -85,B 0,C 180,E1 -27026.086,E2 -27026.086} C_VEL
LIN {X 0,Y 150.547,Z 555.306,A -85,B 0,C 180,E1 -27028.222,E2 -27028.222} C_VEL
LIN {X 0,Y 141.451,Z 567.486,A -85,B 0,C 180,E1 -27031.014,E2 -27031.014} C_VEL
LIN {X 0,Y 132.136,Z 578.334,A -85,B 0,C 180,E1 -27034.474,E2 -27034.474} C_VEL
LIN {X 0,Y 123.623,Z 587.228,A -85,B 0,C 180,E1 -27038.409,E2 -27038.409} C_VEL
LIN {X 0,Y 115.547,Z 594.908,A -85,B 0,C 180,E1 -27043.126,E2 -27043.126} C_VEL
LIN {X 0,Y 107.471,Z 601.932,A -85,B 0,C 180,E1 -27049.163,E2 -27049.163} C_VEL
LIN {X 0,Y 100.774,Z 607.468,A -85,B 0,C 180,E1 -27056.09,E2 -27056.09} C_VEL
LIN {X 0,Y 95.703,Z 611.67,A -85,B 0,C 180,E1 -27063.859,E2 -27063.859} C_VEL
LIN {X 0,Y 92.383,Z 614.63,A -85,B 0,C 180,E1 -27072.286,E2 -27072.286} C_VEL
LIN {X 0,Y 90.986,Z 616.416,A -85,B 0,C 180,E1 -27081.115,E2 -27081.115} C_VEL
LIN {X 0,Y 91.105,Z 617.044,A -85,B 0,C 180,E1 -27090.002,E2 -27090.002} C_VEL
LIN {X 0,Y 90.986,Z 616.395,A -85,B 0,C 180,E1 -27098.889,E2 -27098.889} C_VEL
LIN {X 0,Y 92.384,Z 614.582,A -85,B 0,C 180,E1 -27107.718,E2 -27107.718} C_VEL
LIN {X 0,Y 95.71,Z 611.599,A -85,B 0,C 180,E1 -27116.143,E2 -27116.143} C_VEL
LIN {X 0,Y 101.056,Z 607.142,A -85,B 0,C 180,E1 -27124.252,E2 -27124.252} C_VEL
LIN {X 0,Y 102.911,Z 605.175,A -85,B 0,C 180,E1 -27127.19,E2 -27127.19} C_VEL
LIN {X 0,Y 106.832,Z 598.493,A -85,B 0,C 180,E1 -27135.987,E2 -27135.987} C_VEL
LIN {X 0,Y 109.173,Z 595.867,A -85,B 0,C 180,E1 -27138.519,E2 -27138.519} C_VEL
LIN {X 0,Y 110.2,Z 594.923,A -85,B 0,C 180,E1 -27139.259,E2 -27139.259} C_VEL
LIN {X 0,Y 119.111,Z 586.924,A -85,B 0,C 180,E1 -27144.225,E2 -27144.225} C_VEL
LIN {X 0,Y 128.233,Z 577.845,A -85,B 0,C 180,E1 -27148.161,E2 -27148.161} C_VEL
LIN {X 0,Y 137.898,Z 566.941,A -85,B 0,C 180,E1 -27151.543,E2 -27151.543} C_VEL
LIN {X 0,Y 146.564,Z 555.728,A -85,B 0,C 180,E1 -27154.043,E2 -27154.043} C_VEL
LIN {X 0,Y 154.697,Z 543.44,A -85,B 0,C 180,E1 -27156.109,E2 -27156.109} C_VEL
LIN {X 0,Y 162.282,Z 529.929,A -85,B 0,C 180,E1 -27157.777,E2 -27157.777} C_VEL
LIN {X 0,Y 168.444,Z 516.653,A -85,B 0,C 180,E1 -27159,E2 -27159} C_VEL
LIN {X 0,Y 173.967,Z 502.127,A -85,B 0,C 180,E1 -27159.933,E2 -27159.933} C_VEL
LIN {X 0,Y 178.294,Z 487.047,A -85,B 0,C 180,E1 -27160.664,E2 -27160.664} C_VEL
LIN {X 0,Y 181.188,Z 472.574,A -85,B 0,C 180,E1 -27161.176,E2 -27161.176} C_VEL
LIN {X 0,Y 184.102,Z 447.922,A -85,B 0,C 180,E1 -27161.755,E2 -27161.755} C_VEL
LIN {X 0,Y 185.622,Z 433.421,A -85,B 0,C 180,E1 -27162.087,E2 -27162.087} C_VEL
LIN {X 0,Y 183.992,Z 427.647,A -85,B 0,C 180,E1 -27164.492,E2 -27164.492} C_VEL
LIN {X 0,Y 182.198,Z 423.469,A -85,B 0,C 180,E1 -27167.327,E2 -27167.327} C_VEL
LIN {X 0,Y 180.871,Z 420.473,A -85,B 0,C 180,E1 -27169.93,E2 -27169.93} C_VEL
LIN {X 0,Y 179.942,Z 418.108,A -85,B 0,C 180,E1 -27172.341,E2 -27172.341} C_VEL
LIN {X 0,Y 178.761,Z 414.353,A -85,B 0,C 180,E1 -27178.504,E2 -27178.504} C_VEL
LIN {X 0,Y 178.791,Z 414.519,A -85,B 0,C 180,E1 -27182.535,E2 -27182.535} C_VEL
LIN {X 0,Y 179.796,Z 417.985,A -85,B 0,C 180,E1 -27187.864,E2 -27187.864} C_VEL
LIN {X 0,Y 181.493,Z 421.863,A -85,B 0,C 180,E1 -27191.945,E2 -27191.945} C_VEL
LIN {X 0,Y 183.621,Z 426.725,A -85,B 0,C 180,E1 -27195.541,E2 -27195.541} C_VEL
LIN {X 0,Y 185.683,Z 431.817,A -85,B 0,C 180,E1 -27198.355,E2 -27198.355} C_VEL
LIN {X 0,Y 181.922,Z 466.435,A -85,B 0,C 180,E1 -27199.237,E2 -27199.237} C_VEL
LIN {X 0,Y 179.014,Z 481.56,A -85,B 0,C 180,E1 -27199.776,E2 -27199.776} C_VEL
LIN {X 0,Y 174.998,Z 496.237,A -85,B 0,C 180,E1 -27200.567,E2 -27200.567} C_VEL
LIN {X 0,Y 170.072,Z 510.012,A -85,B 0,C 180,E1 -27201.596,E2 -27201.596} C_VEL
LIN {X 0,Y 163.955,Z 523.839,A -85,B 0,C 180,E1 -27202.992,E2 -27202.992} C_VEL
LIN {X 0,Y 156.743,Z 537.243,A -85,B 0,C 180,E1 -27204.771,E2 -27204.771} C_VEL
LIN {X 0,Y 148.696,Z 549.63,A -85,B 0,C 180,E1 -27206.857,E2 -27206.857} C_VEL
LIN {X 0,Y 140.855,Z 559.999,A -85,B 0,C 180,E1 -27209.168,E2 -27209.168} C_VEL
LIN {X 0,Y 132.691,Z 569.607,A -85,B 0,C 180,E1 -27212.062,E2 -27212.062} C_VEL
LIN {X 0,Y 124.945,Z 577.797,A -85,B 0,C 180,E1 -27215.349,E2 -27215.349} C_VEL
LIN {X 0,Y 116.279,Z 585.854,A -85,B 0,C 180,E1 -27219.587,E2 -27219.587} C_VEL
LIN {X 0,Y 108.356,Z 592.496,A -85,B 0,C 180,E1 -27224.48,E2 -27224.48} C_VEL
LIN {X 0,Y 100.379,Z 598.631,A -85,B 0,C 180,E1 -27230.937,E2 -27230.937} C_VEL
LIN {X 0,Y 93.803,Z 603.356,A -85,B 0,C 180,E1 -27238.365,E2 -27238.365} C_VEL
LIN {X 0,Y 88.785,Z 606.807,A -85,B 0,C 180,E1 -27246.682,E2 -27246.682} C_VEL
LIN {X 0,Y 85.621,Z 609.074,A -85,B 0,C 180,E1 -27255.742,E2 -27255.742} C_VEL
LIN {X 0,Y 84.238,Z 610.218,A -85,B 0,C 180,E1 -27265.212,E2 -27265.212} C_VEL
LIN {X 0,Y 84.141,Z 610.368,A -85,B 0,C 180,E1 -27269.998,E2 -27269.998} C_VEL
LIN {X 0,Y 84.735,Z 609.813,A -85,B 0,C 180,E1 -27279.546,E2 -27279.546} C_VEL
LIN {X 0,Y 86.954,Z 608.154,A -85,B 0,C 180,E1 -27288.86,E2 -27288.86} C_VEL
LIN {X 0,Y 90.976,Z 605.343,A -85,B 0,C 180,E1 -27297.611,E2 -27297.611} C_VEL
LIN {X 0,Y 96.866,Z 601.3,A -85,B 0,C 180,E1 -27305.478,E2 -27305.478} C_VEL
LIN {X 0,Y 104.126,Z 595.936,A -85,B 0,C 180,E1 -27312.448,E2 -27312.448} C_VEL
LIN {X 0,Y 112.71,Z 589.085,A -85,B 0,C 180,E1 -27318.437,E2 -27318.437} C_VEL
LIN {X 0,Y 122.282,Z 580.526,A -85,B 0,C 180,E1 -27323.572,E2 -27323.572} C_VEL
LIN {X 0,Y 128.456,Z 574.438,A -85,B 0,C 180,E1 -27326.258,E2 -27326.258} C_VEL
LIN {X 0,Y 135.281,Z 566.984,A -85,B 0,C 180,E1 -27329.001,E2 -27329.001} C_VEL
LIN {X 0,Y 143.652,Z 556.856,A -85,B 0,C 180,E1 -27331.716,E2 -27331.716} C_VEL
LIN {X 0,Y 152.233,Z 544.789,A -85,B 0,C 180,E1 -27334.186,E2 -27334.186} C_VEL
LIN {X 0,Y 159.592,Z 532.678,A -85,B 0,C 180,E1 -27336.03,E2 -27336.03} C_VEL
LIN {X 0,Y 166.138,Z 519.71,A -85,B 0,C 180,E1 -27337.621,E2 -27337.621} C_VEL
LIN {X 0,Y 171.509,Z 506.946,A -85,B 0,C 180,E1 -27338.784,E2 -27338.784} C_VEL
LIN {X 0,Y 176.474,Z 492.209,A -85,B 0,C 180,E1 -27339.776,E2 -27339.776} C_VEL
LIN {X 0,Y 180.226,Z 477.093,A -85,B 0,C 180,E1 -27340.536,E2 -27340.536} C_VEL
LIN {X 0,Y 182.721,Z 462.114,A -85,B 0,C 180,E1 -27341.038,E2 -27341.038} C_VEL
LIN {X 0,Y 185.935,Z 431.937,A -85,B 0,C 180,E1 -27341.771,E2 -27341.771} C_VEL
LIN {X 0,Y 183.381,Z 425.855,A -85,B 0,C 180,E1 -27345.327,E2 -27345.327} C_VEL
LIN {X 0,Y 181.301,Z 421.114,A -85,B 0,C 180,E1 -27349.107,E2 -27349.107} C_VEL
LIN {X 0,Y 180.116,Z 418.24,A -85,B 0,C 180,E1 -27352.15,E2 -27352.15} C_VEL
LIN {X 0,Y 179.058,Z 414.426,A -85,B 0,C 180,E1 -27358.313,E2 -27358.313} C_VEL
LIN {X 0,Y 179.059,Z 414.662,A -85,B 0,C 180,E1 -27361.546,E2 -27361.546} C_VEL
LIN {X 0,Y 180.382,Z 418.805,A -85,B 0,C 180,E1 -27368.119,E2 -27368.119} C_VEL
LIN {X 0,Y 181.948,Z 422.511,A -85,B 0,C 180,E1 -27371.7,E2 -27371.7} C_VEL
LIN {X 0,Y 183.713,Z 426.532,A -85,B 0,C 180,E1 -27374.681,E2 -27374.681} C_VEL
LIN {X 0,Y 184.767,Z 429.587,A -85,B 0,C 180,E1 -27376.276,E2 -27376.276} C_VEL
LIN {X 0,Y 185.849,Z 433.571,A -85,B 0,C 180,E1 -27377.856,E2 -27377.856} C_VEL
LIN {X 0,Y 181.656,Z 471.441,A -85,B 0,C 180,E1 -27378.763,E2 -27378.763} C_VEL
LIN {X 0,Y 178.679,Z 486.527,A -85,B 0,C 180,E1 -27379.269,E2 -27379.269} C_VEL
LIN {X 0,Y 174.376,Z 501.745,A -85,B 0,C 180,E1 -27380.021,E2 -27380.021} C_VEL
LIN {X 0,Y 169.257,Z 515.465,A -85,B 0,C 180,E1 -27380.894,E2 -27380.894} C_VEL
LIN {X 0,Y 163.061,Z 528.914,A -85,B 0,C 180,E1 -27382.083,E2 -27382.083} C_VEL
LIN {X 0,Y 155.448,Z 542.616,A -85,B 0,C 180,E1 -27383.722,E2 -27383.722} C_VEL
LIN {X 0,Y 147.3,Z 555.037,A -85,B 0,C 180,E1 -27385.77,E2 -27385.77} C_VEL
LIN {X 0,Y 137.915,Z 567.217,A -85,B 0,C 180,E1 -27388.476,E2 -27388.476} C_VEL
LIN {X 0,Y 128.232,Z 578.064,A -85,B 0,C 180,E1 -27391.845,E2 -27391.845} C_VEL
LIN {X 0,Y 119.018,Z 587.213,A -85,B 0,C 180,E1 -27395.844,E2 -27395.844} C_VEL
LIN {X 0,Y 110.738,Z 594.635,A -85,B 0,C 180,E1 -27400.399,E2 -27400.399} C_VEL
LIN {X 0,Y 102.137,Z 601.659,A -85,B 0,C 180,E1 -27406.523,E2 -27406.523} C_VEL
LIN {X 0,Y 94.901,Z 607.196,A -85,B 0,C 180,E1 -27413.671,E2 -27413.671} C_VEL
LIN {X 0,Y 89.313,Z 611.397,A -85,B 0,C 180,E1 -27421.829,E2 -27421.829} C_VEL
LIN {X 0,Y 85.578,Z 614.357,A -85,B 0,C 180,E1 -27430.825,E2 -27430.825} C_VEL
LIN {X 0,Y 83.948,Z 616.144,A -85,B 0,C 180,E1 -27440.363,E2 -27440.363} C_VEL
LIN {X 0,Y 84.01,Z 616.774,A -85,B 0,C 180,E1 -27450.002,E2 -27450.002} C_VEL
LIN {X 0,Y 83.948,Z 616.123,A -85,B 0,C 180,E1 -27459.641,E2 -27459.641} C_VEL
LIN {X 0,Y 85.579,Z 614.308,A -85,B 0,C 180,E1 -27469.18,E2 -27469.18} C_VEL
LIN {X 0,Y 89.323,Z 611.325,A -85,B 0,C 180,E1 -27478.172,E2 -27478.172} C_VEL
LIN {X 0,Y 94.905,Z 607.101,A -85,B 0,C 180,E1 -27486.332,E2 -27486.332} C_VEL
LIN {X 0,Y 102.111,Z 601.529,A -85,B 0,C 180,E1 -27493.496,E2 -27493.496} C_VEL
LIN {X 0,Y 110.2,Z 594.923,A -85,B 0,C 180,E1 -27499.259,E2 -27499.259} C_VEL
LIN {X 0,Y 113.008,Z 592.099,A -85,B 0,C 180,E1 -27501.505,E2 -27501.505} C_VEL
LIN {X 0,Y 119.541,Z 583.058,A -85,B 0,C 180,E1 -27508.378,E2 -27508.378} C_VEL
LIN {X 0,Y 122.521,Z 579.638,A -85,B 0,C 180,E1 -27510.165,E2 -27510.165} C_VEL
LIN {X 0,Y 123.712,Z 578.437,A -85,B 0,C 180,E1 -27510.638,E2 -27510.638} C_VEL
LIN {X 0,Y 133.171,Z 568.31,A -85,B 0,C 180,E1 -27513.791,E2 -27513.791} C_VEL
LIN {X 0,Y 142.09,Z 557.415,A -85,B 0,C 180,E1 -27516.215,E2 -27516.215} C_VEL
LIN {X 0,Y 150.394,Z 545.573,A -85,B 0,C 180,E1 -27518.209,E2 -27518.209} C_VEL
LIN {X 0,Y 158.157,Z 532.517,A -85,B 0,C 180,E1 -27519.843,E2 -27519.843} C_VEL
LIN {X 0,Y 165.235,Z 518.147,A -85,B 0,C 180,E1 -27521.154,E2 -27521.154} C_VEL
LIN {X 0,Y 170.86,Z 504.11,A -85,B 0,C 180,E1 -27522.031,E2 -27522.031} C_VEL
LIN {X 0,Y 175.469,Z 489.057,A -85,B 0,C 180,E1 -27522.752,E2 -27522.752} C_VEL
LIN {X 0,Y 178.721,Z 474.019,A -85,B 0,C 180,E1 -27523.28,E2 -27523.28} C_VEL
LIN {X 0,Y 181.178,Z 455.333,A -85,B 0,C 180,E1 -27523.707,E2 -27523.707} C_VEL
LIN {X 0,Y 183.156,Z 436.893,A -85,B 0,C 180,E1 -27524.117,E2 -27524.117} C_VEL
LIN {X 0,Y 182.123,Z 433.159,A -85,B 0,C 180,E1 -27525.845,E2 -27525.845} C_VEL
LIN {X 0,Y 180.696,Z 429.671,A -85,B 0,C 180,E1 -27528.36,E2 -27528.36} C_VEL
LIN {X 0,Y 179.512,Z 426.746,A -85,B 0,C 180,E1 -27530.991,E2 -27530.991} C_VEL
LIN {X 0,Y 178.754,Z 424.753,A -85,B 0,C 180,E1 -27533.226,E2 -27533.226} C_VEL
LIN {X 0,Y 177.894,Z 421.419,A -85,B 0,C 180,E1 -27538.497,E2 -27538.497} C_VEL
LIN {X 0,Y 177.897,Z 421.538,A -85,B 0,C 180,E1 -27542.264,E2 -27542.264} C_VEL
LIN {X 0,Y 179.072,Z 425.671,A -85,B 0,C 180,E1 -27548.393,E2 -27548.393} C_VEL
LIN {X 0,Y 180.551,Z 429.35,A -85,B 0,C 180,E1 -27551.939,E2 -27551.939} C_VEL
LIN {X 0,Y 182.415,Z 434.01,A -85,B 0,C 180,E1 -27555.217,E2 -27555.217} C_VEL
LIN {X 0,Y 183.124,Z 435.843,A -85,B 0,C 180,E1 -27556.284,E2 -27556.284} C_VEL
LIN {X 0,Y 182.165,Z 445.527,A -85,B 0,C 180,E1 -27556.586,E2 -27556.586} C_VEL
LIN {X 0,Y 179.447,Z 468.214,A -85,B 0,C 180,E1 -27557.142,E2 -27557.142} C_VEL
LIN {X 0,Y 176.547,Z 482.606,A -85,B 0,C 180,E1 -27557.65,E2 -27557.65} C_VEL
LIN {X 0,Y 172.25,Z 497.663,A -85,B 0,C 180,E1 -27558.441,E2 -27558.441} C_VEL
LIN {X 0,Y 166.823,Z 512.141,A -85,B 0,C 180,E1 -27559.499,E2 -27559.499} C_VEL
LIN {X 0,Y 160.659,Z 525.438,A -85,B 0,C 180,E1 -27560.82,E2 -27560.82} C_VEL
LIN {X 0,Y 153.139,Z 538.753,A -85,B 0,C 180,E1 -27562.538,E2 -27562.538} C_VEL
LIN {X 0,Y 144.879,Z 550.937,A -85,B 0,C 180,E1 -27564.553,E2 -27564.553} C_VEL
LIN {X 0,Y 136.097,Z 562.034,A -85,B 0,C 180,E1 -27567.024,E2 -27567.024} C_VEL
LIN {X 0,Y 126.968,Z 572.135,A -85,B 0,C 180,E1 -27570.177,E2 -27570.177} C_VEL
LIN {X 0,Y 119.616,Z 579.292,A -85,B 0,C 180,E1 -27573.146,E2 -27573.146} C_VEL
LIN {X 0,Y 110.626,Z 587.125,A -85,B 0,C 180,E1 -27577.425,E2 -27577.425} C_VEL
LIN {X 0,Y 101.221,Z 594.43,A -85,B 0,C 180,E1 -27583.191,E2 -27583.191} C_VEL
LIN {X 0,Y 93.02,Z 600.211,A -85,B 0,C 180,E1 -27590.041,E2 -27590.041} C_VEL
LIN {X 0,Y 87.833,Z 603.628,A -85,B 0,C 180,E1 -27595.934,E2 -27595.934} C_VEL
LIN {X 0,Y 82.291,Z 607.079,A -85,B 0,C 180,E1 -27604.719,E2 -27604.719} C_VEL
LIN {X 0,Y 78.757,Z 609.344,A -85,B 0,C 180,E1 -27614.469,E2 -27614.469} C_VEL
LIN {X 0,Y 77.172,Z 610.488,A -85,B 0,C 180,E1 -27624.772,E2 -27624.772} C_VEL
LIN {X 0,Y 77.06,Z 610.637,A -85,B 0,C 180,E1 -27629.997,E2 -27629.997} C_VEL
LIN {X 0,Y 77.735,Z 610.083,A -85,B 0,C 180,E1 -27640.415,E2 -27640.415} C_VEL
LIN {X 0,Y 80.259,Z 608.424,A -85,B 0,C 180,E1 -27650.501,E2 -27650.501} C_VEL
LIN {X 0,Y 84.722,Z 605.614,A -85,B 0,C 180,E1 -27659.847,E2 -27659.847} C_VEL
LIN {X 0,Y 91.143,Z 601.571,A -85,B 0,C 180,E1 -27668.086,E2 -27668.086} C_VEL
LIN {X 0,Y 98.971,Z 596.207,A -85,B 0,C 180,E1 -27675.241,E2 -27675.241} C_VEL
LIN {X 0,Y 108.113,Z 589.355,A -85,B 0,C 180,E1 -27681.265,E2 -27681.265} C_VEL
LIN {X 0,Y 118.208,Z 580.794,A -85,B 0,C 180,E1 -27686.339,E2 -27686.339} C_VEL
LIN {X 0,Y 125.229,Z 574.089,A -85,B 0,C 180,E1 -27689.259,E2 -27689.259} C_VEL
LIN {X 0,Y 134.592,Z 564.025,A -85,B 0,C 180,E1 -27692.582,E2 -27692.582} C_VEL
LIN {X 0,Y 143.349,Z 553.307,A -85,B 0,C 180,E1 -27695.091,E2 -27695.091} C_VEL
LIN {X 0,Y 151.529,Z 541.603,A -85,B 0,C 180,E1 -27697.189,E2 -27697.189} C_VEL
LIN {X 0,Y 159.244,Z 528.578,A -85,B 0,C 180,E1 -27698.941,E2 -27698.941} C_VEL
LIN {X 0,Y 165.196,Z 516.449,A -85,B 0,C 180,E1 -27700.264,E2 -27700.264} C_VEL
LIN {X 0,Y 170.636,Z 503.152,A -85,B 0,C 180,E1 -27701.314,E2 -27701.314} C_VEL
LIN {X 0,Y 175.34,Z 488.483,A -85,B 0,C 180,E1 -27702.164,E2 -27702.164} C_VEL
LIN {X 0,Y 178.807,Z 473.431,A -85,B 0,C 180,E1 -27702.839,E2 -27702.839} C_VEL
LIN {X 0,Y 181.113,Z 458.033,A -85,B 0,C 180,E1 -27703.246,E2 -27703.246} C_VEL
LIN {X 0,Y 183.413,Z 436.137,A -85,B 0,C 180,E1 -27703.785,E2 -27703.785} C_VEL
LIN {X 0,Y 181.312,Z 430.752,A -85,B 0,C 180,E1 -27707.228,E2 -27707.228} C_VEL
LIN {X 0,Y 179.919,Z 427.444,A -85,B 0,C 180,E1 -27710.16,E2 -27710.16} C_VEL
LIN {X 0,Y 178.971,Z 424.931,A -85,B 0,C 180,E1 -27712.951,E2 -27712.951} C_VEL
LIN {X 0,Y 178.159,Z 421.452,A -85,B 0,C 180,E1 -27718.87,E2 -27718.87} C_VEL
LIN {X 0,Y 178.173,Z 421.776,A -85,B 0,C 180,E1 -27721.412,E2 -27721.412} C_VEL
LIN {X 0,Y 179.328,Z 425.754,A -85,B 0,C 180,E1 -27727.692,E2 -27727.692} C_VEL
LIN {X 0,Y 180.704,Z 429.229,A -85,B 0,C 180,E1 -27731.083,E2 -27731.083} C_VEL
LIN {X 0,Y 182.393,Z 433.43,A -85,B 0,C 180,E1 -27734.148,E2 -27734.148} C_VEL
LIN {X 0,Y 183.36,Z 436.919,A -85,B 0,C 180,E1 -27735.775,E2 -27735.775} C_VEL
LIN {X 0,Y 182.948,Z 441.471,A -85,B 0,C 180,E1 -27735.958,E2 -27735.958} C_VEL
LIN {X 0,Y 179.418,Z 471.668,A -85,B 0,C 180,E1 -27736.634,E2 -27736.634} C_VEL
LIN {X 0,Y 176.263,Z 487.029,A -85,B 0,C 180,E1 -27737.124,E2 -27737.124} C_VEL
LIN {X 0,Y 172.068,Z 501.481,A -85,B 0,C 180,E1 -27737.793,E2 -27737.793} C_VEL
LIN {X 0,Y 166.854,Z 515.2,A -85,B 0,C 180,E1 -27738.613,E2 -27738.613} C_VEL
LIN {X 0,Y 160.516,Z 528.647,A -85,B 0,C 180,E1 -27739.723,E2 -27739.723} C_VEL
LIN {X 0,Y 152.718,Z 542.348,A -85,B 0,C 180,E1 -27741.271,E2 -27741.271} C_VEL
LIN {X 0,Y 144.347,Z 554.769,A -85,B 0,C 180,E1 -27743.224,E2 -27743.224} C_VEL
LIN {X 0,Y 134.664,Z 566.948,A -85,B 0,C 180,E1 -27745.811,E2 -27745.811} C_VEL
LIN {X 0,Y 126.014,Z 576.359,A -85,B 0,C 180,E1 -27748.553,E2 -27748.553} C_VEL
LIN {X 0,Y 116.375,Z 585.623,A -85,B 0,C 180,E1 -27752.28,E2 -27752.28} C_VEL
LIN {X 0,Y 106.225,Z 594.363,A -85,B 0,C 180,E1 -27757.448,E2 -27757.448} C_VEL
LIN {X 0,Y 97.049,Z 601.386,A -85,B 0,C 180,E1 -27763.603,E2 -27763.603} C_VEL
LIN {X 0,Y 89.21,Z 606.923,A -85,B 0,C 180,E1 -27770.935,E2 -27770.935} C_VEL
LIN {X 0,Y 83.057,Z 611.125,A -85,B 0,C 180,E1 -27779.492,E2 -27779.492} C_VEL
LIN {X 0,Y 78.838,Z 614.085,A -85,B 0,C 180,E1 -27789.112,E2 -27789.112} C_VEL
LIN {X 0,Y 76.913,Z 615.872,A -85,B 0,C 180,E1 -27799.472,E2 -27799.472} C_VEL
LIN {X 0,Y 76.906,Z 616.503,A -85,B 0,C 180,E1 -27810.003,E2 -27810.003} C_VEL
LIN {X 0,Y 76.914,Z 615.851,A -85,B 0,C 180,E1 -27820.533,E2 -27820.533} C_VEL
LIN {X 0,Y 78.839,Z 614.035,A -85,B 0,C 180,E1 -27830.893,E2 -27830.893} C_VEL
LIN {X 0,Y 83.071,Z 611.051,A -85,B 0,C 180,E1 -27840.508,E2 -27840.508} C_VEL
LIN {X 0,Y 89.212,Z 606.826,A -85,B 0,C 180,E1 -27849.07,E2 -27849.07} C_VEL
LIN {X 0,Y 97.026,Z 601.255,A -85,B 0,C 180,E1 -27856.417,E2 -27856.417} C_VEL
LIN {X 0,Y 106.224,Z 594.191,A -85,B 0,C 180,E1 -27862.559,E2 -27862.559} C_VEL
LIN {X 0,Y 115.07,Z 586.649,A -85,B 0,C 180,E1 -27867.12,E2 -27867.12} C_VEL
LIN {X 0,Y 123.712,Z 578.437,A -85,B 0,C 180,E1 -27870.638,E2 -27870.638} C_VEL
LIN {X 0,Y 127.028,Z 574.812,A -85,B 0,C 180,E1 -27872.131,E2 -27872.131} C_VEL
LIN {X 0,Y 131.372,Z 568.691,A -85,B 0,C 180,E1 -27874.995,E2 -27874.995} C_VEL
LIN {X 0,Y 135.65,Z 562.189,A -85,B 0,C 180,E1 -27877.629,E2 -27877.629} C_VEL
LIN {X 0,Y 138.749,Z 557.921,A -85,B 0,C 180,E1 -27878.757,E2 -27878.757} C_VEL
LIN {X 0,Y 147.947,Z 545.198,A -85,B 0,C 180,E1 -27880.803,E2 -27880.803} C_VEL
LIN {X 0,Y 155.849,Z 532.241,A -85,B 0,C 180,E1 -27882.299,E2 -27882.299} C_VEL
LIN {X 0,Y 162.269,Z 519.64,A -85,B 0,C 180,E1 -27883.391,E2 -27883.391} C_VEL
LIN {X 0,Y 168.393,Z 504.962,A -85,B 0,C 180,E1 -27884.27,E2 -27884.27} C_VEL
LIN {X 0,Y 173.085,Z 490.303,A -85,B 0,C 180,E1 -27884.937,E2 -27884.937} C_VEL
LIN {X 0,Y 176.466,Z 475.633,A -85,B 0,C 180,E1 -27885.44,E2 -27885.44} C_VEL
LIN {X 0,Y 178.726,Z 460.365,A -85,B 0,C 180,E1 -27885.779,E2 -27885.779} C_VEL
LIN {X 0,Y 180.887,Z 440.448,A -85,B 0,C 180,E1 -27886.233,E2 -27886.233} C_VEL
LIN {X 0,Y 179.58,Z 436.713,A -85,B 0,C 180,E1 -27888.716,E2 -27888.716} C_VEL
LIN {X 0,Y 178.357,Z 433.44,A -85,B 0,C 180,E1 -27891.645,E2 -27891.645} C_VEL
LIN {X 0,Y 177.71,Z 431.607,A -85,B 0,C 180,E1 -27893.757,E2 -27893.757} C_VEL
LIN {X 0,Y 177,Z 428.429,A -85,B 0,C 180,E1 -27898.867,E2 -27898.867} C_VEL
LIN {X 0,Y 177.006,Z 428.571,A -85,B 0,C 180,E1 -27901.991,E2 -27901.991} C_VEL
LIN {X 0,Y 177.976,Z 432.476,A -85,B 0,C 180,E1 -27907.802,E2 -27907.802} C_VEL
LIN {X 0,Y 179.244,Z 435.915,A -85,B 0,C 180,E1 -27911.163,E2 -27911.163} C_VEL
LIN {X 0,Y 180.733,Z 439.92,A -85,B 0,C 180,E1 -27914.066,E2 -27914.066} C_VEL
LIN {X 0,Y 180.868,Z 440.286,A -85,B 0,C 180,E1 -27914.297,E2 -27914.297} C_VEL
LIN {X 0,Y 177.743,Z 467.099,A -85,B 0,C 180,E1 -27914.927,E2 -27914.927} C_VEL
LIN {X 0,Y 174.733,Z 482.12,A -85,B 0,C 180,E1 -27915.404,E2 -27915.404} C_VEL
LIN {X 0,Y 170.533,Z 496.793,A -85,B 0,C 180,E1 -27916.101,E2 -27916.101} C_VEL
LIN {X 0,Y 165.383,Z 510.564,A -85,B 0,C 180,E1 -27917.027,E2 -27917.027} C_VEL
LIN {X 0,Y 159.086,Z 524.12,A -85,B 0,C 180,E1 -27918.255,E2 -27918.255} C_VEL
LIN {X 0,Y 151.353,Z 537.791,A -85,B 0,C 180,E1 -27919.894,E2 -27919.894} C_VEL
LIN {X 0,Y 142.846,Z 550.177,A -85,B 0,C 180,E1 -27921.771,E2 -27921.771} C_VEL
LIN {X 0,Y 134.508,Z 560.546,A -85,B 0,C 180,E1 -27923.88,E2 -27923.88} C_VEL
LIN {X 0,Y 125.325,Z 570.531,A -85,B 0,C 180,E1 -27926.656,E2 -27926.656} C_VEL
LIN {X 0,Y 115.891,Z 579.564,A -85,B 0,C 180,E1 -27930.209,E2 -27930.209} C_VEL
LIN {X 0,Y 106.449,Z 587.398,A -85,B 0,C 180,E1 -27934.38,E2 -27934.38} C_VEL
LIN {X 0,Y 96.487,Z 594.702,A -85,B 0,C 180,E1 -27940.107,E2 -27940.107} C_VEL
LIN {X 0,Y 87.671,Z 600.484,A -85,B 0,C 180,E1 -27947.045,E2 -27947.045} C_VEL
LIN {X 0,Y 82.028,Z 603.9,A -85,B 0,C 180,E1 -27953.145,E2 -27953.145} C_VEL
LIN {X 0,Y 75.916,Z 607.351,A -85,B 0,C 180,E1 -27962.424,E2 -27962.424} C_VEL
LIN {X 0,Y 71.924,Z 609.616,A -85,B 0,C 180,E1 -27972.951,E2 -27972.951} C_VEL
LIN {X 0,Y 70.102,Z 610.758,A -85,B 0,C 180,E1 -27984.243,E2 -27984.243} C_VEL
LIN {X 0,Y 69.969,Z 610.908,A -85,B 0,C 180,E1 -27989.997,E2 -27989.997} C_VEL
LIN {X 0,Y 70.774,Z 610.353,A -85,B 0,C 180,E1 -28001.453,E2 -28001.453} C_VEL
LIN {X 0,Y 73.619,Z 608.695,A -85,B 0,C 180,E1 -28012.446,E2 -28012.446} C_VEL
LIN {X 0,Y 78.619,Z 605.885,A -85,B 0,C 180,E1 -28022.433,E2 -28022.433} C_VEL
LIN {X 0,Y 85.623,Z 601.843,A -85,B 0,C 180,E1 -28031.042,E2 -28031.042} C_VEL
LIN {X 0,Y 94.086,Z 596.477,A -85,B 0,C 180,E1 -28038.326,E2 -28038.326} C_VEL
LIN {X 0,Y 103.809,Z 589.625,A -85,B 0,C 180,E1 -28044.329,E2 -28044.329} C_VEL
LIN {X 0,Y 113.033,Z 582.257,A -85,B 0,C 180,E1 -28048.749,E2 -28048.749} C_VEL
LIN {X 0,Y 120.007,Z 576.047,A -85,B 0,C 180,E1 -28051.452,E2 -28051.452} C_VEL
LIN {X 0,Y 127.072,Z 569.011,A -85,B 0,C 180,E1 -28053.99,E2 -28053.99} C_VEL
LIN {X 0,Y 135.977,Z 559.164,A -85,B 0,C 180,E1 -28056.547,E2 -28056.547} C_VEL
LIN {X 0,Y 145.067,Z 547.451,A -85,B 0,C 180,E1 -28058.84,E2 -28058.84} C_VEL
LIN {X 0,Y 152.821,Z 535.779,A -85,B 0,C 180,E1 -28060.518,E2 -28060.518} C_VEL
LIN {X 0,Y 159.809,Z 523.169,A -85,B 0,C 180,E1 -28062.005,E2 -28062.005} C_VEL
LIN {X 0,Y 166.108,Z 509.455,A -85,B 0,C 180,E1 -28063.185,E2 -28063.185} C_VEL
LIN {X 0,Y 171.295,Z 495.326,A -85,B 0,C 180,E1 -28064.069,E2 -28064.069} C_VEL
LIN {X 0,Y 175.34,Z 480.709,A -85,B 0,C 180,E1 -28064.767,E2 -28064.767} C_VEL
LIN {X 0,Y 178.194,Z 465.861,A -85,B 0,C 180,E1 -28065.261,E2 -28065.261} C_VEL
LIN {X 0,Y 181.13,Z 440.514,A -85,B 0,C 180,E1 -28065.818,E2 -28065.818} C_VEL
LIN {X 0,Y 179.495,Z 436.102,A -85,B 0,C 180,E1 -28068.996,E2 -28068.996} C_VEL
LIN {X 0,Y 178.47,Z 433.392,A -85,B 0,C 180,E1 -28071.615,E2 -28071.615} C_VEL
LIN {X 0,Y 177.938,Z 431.776,A -85,B 0,C 180,E1 -28073.474,E2 -28073.474} C_VEL
LIN {X 0,Y 177.296,Z 428.484,A -85,B 0,C 180,E1 -28078.864,E2 -28078.864} C_VEL
LIN {X 0,Y 177.289,Z 428.784,A -85,B 0,C 180,E1 -28081.135,E2 -28081.135} C_VEL
LIN {X 0,Y 178.311,Z 432.758,A -85,B 0,C 180,E1 -28087.342,E2 -28087.342} C_VEL
LIN {X 0,Y 179.518,Z 436.059,A -85,B 0,C 180,E1 -28090.544,E2 -28090.544} C_VEL
LIN {X 0,Y 180.969,Z 440.013,A -85,B 0,C 180,E1 -28093.403,E2 -28093.403} C_VEL
LIN {X 0,Y 181.149,Z 440.684,A -85,B 0,C 180,E1 -28093.743,E2 -28093.743} C_VEL
LIN {X 0,Y 177.601,Z 470.937,A -85,B 0,C 180,E1 -28094.426,E2 -28094.426} C_VEL
LIN {X 0,Y 174.517,Z 486.006,A -85,B 0,C 180,E1 -28094.874,E2 -28094.874} C_VEL
LIN {X 0,Y 170.037,Z 501.218,A -85,B 0,C 180,E1 -28095.519,E2 -28095.519} C_VEL
LIN {X 0,Y 164.723,Z 514.935,A -85,B 0,C 180,E1 -28096.269,E2 -28096.269} C_VEL
LIN {X 0,Y 158.257,Z 528.381,A -85,B 0,C 180,E1 -28097.298,E2 -28097.298} C_VEL
LIN {X 0,Y 150.273,Z 542.08,A -85,B 0,C 180,E1 -28098.732,E2 -28098.732} C_VEL
LIN {X 0,Y 141.691,Z 554.501,A -85,B 0,C 180,E1 -28100.578,E2 -28100.578} C_VEL
LIN {X 0,Y 131.719,Z 566.679,A -85,B 0,C 180,E1 -28103.02,E2 -28103.02} C_VEL
LIN {X 0,Y 122.757,Z 576.089,A -85,B 0,C 180,E1 -28105.62,E2 -28105.62} C_VEL
LIN {X 0,Y 112.713,Z 585.352,A -85,B 0,C 180,E1 -28109.201,E2 -28109.201} C_VEL
LIN {X 0,Y 104.557,Z 592.115,A -85,B 0,C 180,E1 -28112.946,E2 -28112.946} C_VEL
LIN {X 0,Y 94.613,Z 599.483,A -85,B 0,C 180,E1 -28118.746,E2 -28118.746} C_VEL
LIN {X 0,Y 85.751,Z 605.388,A -85,B 0,C 180,E1 -28125.844,E2 -28125.844} C_VEL
LIN {X 0,Y 80.129,Z 608.911,A -85,B 0,C 180,E1 -28132.126,E2 -28132.126} C_VEL
LIN {X 0,Y 74.315,Z 612.483,A -85,B 0,C 180,E1 -28141.783,E2 -28141.783} C_VEL
LIN {X 0,Y 70.744,Z 614.851,A -85,B 0,C 180,E1 -28152.663,E2 -28152.663} C_VEL
LIN {X 0,Y 69.593,Z 616.062,A -85,B 0,C 180,E1 -28164.207,E2 -28164.207} C_VEL
LIN {X 0,Y 69.809,Z 616.233,A -85,B 0,C 180,E1 -28170.003,E2 -28170.003} C_VEL
LIN {X 0,Y 69.913,Z 615.579,A -85,B 0,C 180,E1 -28181.601,E2 -28181.601} C_VEL
LIN {X 0,Y 72.185,Z 613.761,A -85,B 0,C 180,E1 -28192.923,E2 -28192.923} C_VEL
LIN {X 0,Y 76.982,Z 610.777,A -85,B 0,C 180,E1 -28203.217,E2 -28203.217} C_VEL
LIN {X 0,Y 83.772,Z 606.552,A -85,B 0,C 180,E1 -28212.159,E2 -28212.159} C_VEL
LIN {X 0,Y 92.227,Z 600.98,A -85,B 0,C 180,E1 -28219.647,E2 -28219.647} C_VEL
LIN {X 0,Y 102.023,Z 593.916,A -85,B 0,C 180,E1 -28225.759,E2 -28225.759} C_VEL
LIN {X 0,Y 111.334,Z 586.372,A -85,B 0,C 180,E1 -28230.228,E2 -28230.228} C_VEL
LIN {X 0,Y 121.291,Z 577.295,A -85,B 0,C 180,E1 -28233.916,E2 -28233.916} C_VEL
LIN {X 0,Y 130.184,Z 568.037,A -85,B 0,C 180,E1 -28236.603,E2 -28236.603} C_VEL
LIN {X 0,Y 138.749,Z 557.921,A -85,B 0,C 180,E1 -28238.757,E2 -28238.757} C_VEL
LIN {X 0,Y 141.816,Z 553.59,A -85,B 0,C 180,E1 -28239.814,E2 -28239.814} C_VEL
LIN {X 0,Y 145.985,Z 546.389,A -85,B 0,C 180,E1 -28241.983,E2 -28241.983} C_VEL
LIN {X 0,Y 149.983,Z 538.868,A -85,B 0,C 180,E1 -28243.927,E2 -28243.927} C_VEL
LIN {X 0,Y 152.676,Z 533.988,A -85,B 0,C 180,E1 -28244.648,E2 -28244.648} C_VEL
LIN {X 0,Y 159.557,Z 521.134,A -85,B 0,C 180,E1 -28245.709,E2 -28245.709} C_VEL
LIN {X 0,Y 165.772,Z 506.942,A -85,B 0,C 180,E1 -28246.525,E2 -28246.525} C_VEL
LIN {X 0,Y 170.954,Z 491.548,A -85,B 0,C 180,E1 -28247.191,E2 -28247.191} C_VEL
LIN {X 0,Y 174.596,Z 476.555,A -85,B 0,C 180,E1 -28247.668,E2 -28247.668} C_VEL
LIN {X 0,Y 176.94,Z 461.668,A -85,B 0,C 180,E1 -28247.97,E2 -28247.97} C_VEL
LIN {X 0,Y 178.81,Z 444.834,A -85,B 0,C 180,E1 -28248.334,E2 -28248.334} C_VEL
LIN {X 0,Y 177.433,Z 440.769,A -85,B 0,C 180,E1 -28251.673,E2 -28251.673} C_VEL
LIN {X 0,Y 176.681,Z 438.46,A -85,B 0,C 180,E1 -28254.293,E2 -28254.293} C_VEL
LIN {X 0,Y 176.115,Z 435.437,A -85,B 0,C 180,E1 -28259.241,E2 -28259.241} C_VEL
LIN {X 0,Y 176.119,Z 435.607,A -85,B 0,C 180,E1 -28261.715,E2 -28261.715} C_VEL
LIN {X 0,Y 176.924,Z 439.325,A -85,B 0,C 180,E1 -28267.284,E2 -28267.284} C_VEL
LIN {X 0,Y 178.019,Z 442.573,A -85,B 0,C 180,E1 -28270.485,E2 -28270.485} C_VEL
LIN {X 0,Y 178.77,Z 444.745,A -85,B 0,C 180,E1 -28272.169,E2 -28272.169} C_VEL
LIN {X 0,Y 175.85,Z 468.468,A -85,B 0,C 180,E1 -28272.716,E2 -28272.716} C_VEL
LIN {X 0,Y 172.783,Z 483.164,A -85,B 0,C 180,E1 -28273.172,E2 -28273.172} C_VEL
LIN {X 0,Y 168.303,Z 498.217,A -85,B 0,C 180,E1 -28273.857,E2 -28273.857} C_VEL
LIN {X 0,Y 162.638,Z 512.693,A -85,B 0,C 180,E1 -28274.782,E2 -28274.782} C_VEL
LIN {X 0,Y 155.903,Z 526.475,A -85,B 0,C 180,E1 -28275.996,E2 -28275.996} C_VEL
LIN {X 0,Y 148.285,Z 539.301,A -85,B 0,C 180,E1 -28277.474,E2 -28277.474} C_VEL
LIN {X 0,Y 139.581,Z 551.483,A -85,B 0,C 180,E1 -28279.248,E2 -28279.248} C_VEL
LIN {X 0,Y 130.251,Z 562.581,A -85,B 0,C 180,E1 -28281.441,E2 -28281.441} C_VEL
LIN {X 0,Y 120.511,Z 572.602,A -85,B 0,C 180,E1 -28284.271,E2 -28284.271} C_VEL
LIN {X 0,Y 111.025,Z 581.058,A -85,B 0,C 180,E1 -28287.594,E2 -28287.594} C_VEL
LIN {X 0,Y 102.591,Z 587.672,A -85,B 0,C 180,E1 -28291.091,E2 -28291.091} C_VEL
LIN {X 0,Y 92.06,Z 594.975,A -85,B 0,C 180,E1 -28296.715,E2 -28296.715} C_VEL
LIN {X 0,Y 82.599,Z 600.757,A -85,B 0,C 180,E1 -28303.675,E2 -28303.675} C_VEL
LIN {X 0,Y 76.437,Z 604.173,A -85,B 0,C 180,E1 -28309.935,E2 -28309.935} C_VEL
LIN {X 0,Y 69.672,Z 607.623,A -85,B 0,C 180,E1 -28319.708,E2 -28319.708} C_VEL
LIN {X 0,Y 65.164,Z 609.887,A -85,B 0,C 180,E1 -28331.119,E2 -28331.119} C_VEL
LIN {X 0,Y 63.063,Z 611.028,A -85,B 0,C 180,E1 -28343.598,E2 -28343.598} C_VEL
LIN {X 0,Y 62.887,Z 611.177,A -85,B 0,C 180,E1 -28349.997,E2 -28349.997} C_VEL
LIN {X 0,Y 63.814,Z 610.624,A -85,B 0,C 180,E1 -28362.722,E2 -28362.722} C_VEL
LIN {X 0,Y 67.092,Z 608.966,A -85,B 0,C 180,E1 -28374.769,E2 -28374.769} C_VEL
LIN {X 0,Y 72.702,Z 606.156,A -85,B 0,C 180,E1 -28385.448,E2 -28385.448} C_VEL
LIN {X 0,Y 80.366,Z 602.114,A -85,B 0,C 180,E1 -28394.391,E2 -28394.391} C_VEL
LIN {X 0,Y 89.503,Z 596.747,A -85,B 0,C 180,E1 -28401.738,E2 -28401.738} C_VEL
LIN {X 0,Y 99.819,Z 589.895,A -85,B 0,C 180,E1 -28407.657,E2 -28407.657} C_VEL
LIN {X 0,Y 109.515,Z 582.526,A -85,B 0,C 180,E1 -28411.929,E2 -28411.929} C_VEL
LIN {X 0,Y 116.755,Z 576.317,A -85,B 0,C 180,E1 -28414.541,E2 -28414.541} C_VEL
LIN {X 0,Y 125.624,Z 567.79,A -85,B 0,C 180,E1 -28417.378,E2 -28417.378} C_VEL
LIN {X 0,Y 134.862,Z 557.66,A -85,B 0,C 180,E1 -28419.719,E2 -28419.719} C_VEL
LIN {X 0,Y 144.237,Z 545.591,A -85,B 0,C 180,E1 -28421.828,E2 -28421.828} C_VEL
LIN {X 0,Y 152.194,Z 533.476,A -85,B 0,C 180,E1 -28423.37,E2 -28423.37} C_VEL
LIN {X 0,Y 159.216,Z 520.59,A -85,B 0,C 180,E1 -28424.707,E2 -28424.707} C_VEL
LIN {X 0,Y 165.009,Z 507.737,A -85,B 0,C 180,E1 -28425.683,E2 -28425.683} C_VEL
LIN {X 0,Y 170.304,Z 492.993,A -85,B 0,C 180,E1 -28426.494,E2 -28426.494} C_VEL
LIN {X 0,Y 174.261,Z 478.02,A -85,B 0,C 180,E1 -28427.139,E2 -28427.139} C_VEL
LIN {X 0,Y 177.067,Z 462.071,A -85,B 0,C 180,E1 -28427.577,E2 -28427.577} C_VEL
LIN {X 0,Y 179.015,Z 445.369,A -85,B 0,C 180,E1 -28427.907,E2 -28427.907} C_VEL
LIN {X 0,Y 178.9,Z 444.565,A -85,B 0,C 180,E1 -28428.241,E2 -28428.241} C_VEL
LIN {X 0,Y 177.643,Z 440.956,A -85,B 0,C 180,E1 -28431.367,E2 -28431.367} C_VEL
LIN {X 0,Y 176.897,Z 438.576,A -85,B 0,C 180,E1 -28434.099,E2 -28434.099} C_VEL
LIN {X 0,Y 176.412,Z 435.683,A -85,B 0,C 180,E1 -28438.858,E2 -28438.858} C_VEL
LIN {X 0,Y 176.416,Z 435.654,A -85,B 0,C 180,E1 -28440.642,E2 -28440.642} C_VEL
LIN {X 0,Y 177.259,Z 439.607,A -85,B 0,C 180,E1 -28446.831,E2 -28446.831} C_VEL
LIN {X 0,Y 178.226,Z 442.547,A -85,B 0,C 180,E1 -28449.699,E2 -28449.699} C_VEL
LIN {X 0,Y 179.098,Z 445.066,A -85,B 0,C 180,E1 -28451.67,E2 -28451.67} C_VEL
LIN {X 0,Y 175.819,Z 471.502,A -85,B 0,C 180,E1 -28452.209,E2 -28452.209} C_VEL
LIN {X 0,Y 172.62,Z 486.508,A -85,B 0,C 180,E1 -28452.619,E2 -28452.619} C_VEL
LIN {X 0,Y 168.275,Z 500.955,A -85,B 0,C 180,E1 -28453.188,E2 -28453.188} C_VEL
LIN {X 0,Y 162.876,Z 514.671,A -85,B 0,C 180,E1 -28453.87,E2 -28453.87} C_VEL
LIN {X 0,Y 156.286,Z 528.115,A -85,B 0,C 180,E1 -28454.803,E2 -28454.803} C_VEL
LIN {X 0,Y 148.145,Z 541.813,A -85,B 0,C 180,E1 -28456.128,E2 -28456.128} C_VEL
LIN {X 0,Y 139.342,Z 554.233,A -85,B 0,C 180,E1 -28457.828,E2 -28457.828} C_VEL
LIN {X 0,Y 129.095,Z 566.41,A -85,B 0,C 180,E1 -28460.103,E2 -28460.103} C_VEL
LIN {X 0,Y 119.838,Z 575.819,A -85,B 0,C 180,E1 -28462.534,E2 -28462.534} C_VEL
LIN {X 0,Y 109.384,Z 585.08,A -85,B 0,C 180,E1 -28465.91,E2 -28465.91} C_VEL
LIN {X 0,Y 100.47,Z 592.112,A -85,B 0,C 180,E1 -28469.69,E2 -28469.69} C_VEL
LIN {X 0,Y 90.294,Z 599.211,A -85,B 0,C 180,E1 -28475.191,E2 -28475.191} C_VEL
LIN {X 0,Y 80.746,Z 605.115,A -85,B 0,C 180,E1 -28482.287,E2 -28482.287} C_VEL
LIN {X 0,Y 74.151,Z 608.901,A -85,B 0,C 180,E1 -28489.308,E2 -28489.308} C_VEL
LIN {X 0,Y 68.078,Z 612.211,A -85,B 0,C 180,E1 -28498.927,E2 -28498.927} C_VEL
LIN {X 0,Y 63.952,Z 614.578,A -85,B 0,C 180,E1 -28510.754,E2 -28510.754} C_VEL
LIN {X 0,Y 62.517,Z 615.79,A -85,B 0,C 180,E1 -28523.548,E2 -28523.548} C_VEL
LIN {X 0,Y 62.702,Z 615.962,A -85,B 0,C 180,E1 -28530.003,E2 -28530.003} C_VEL
LIN {X 0,Y 62.919,Z 615.306,A -85,B 0,C 180,E1 -28542.912,E2 -28542.912} C_VEL
LIN {X 0,Y 65.645,Z 613.488,A -85,B 0,C 180,E1 -28555.36,E2 -28555.36} C_VEL
LIN {X 0,Y 71.099,Z 610.504,A -85,B 0,C 180,E1 -28566.38,E2 -28566.38} C_VEL
LIN {X 0,Y 78.591,Z 606.278,A -85,B 0,C 180,E1 -28575.68,E2 -28575.68} C_VEL
LIN {X 0,Y 87.75,Z 600.705,A -85,B 0,C 180,E1 -28583.221,E2 -28583.221} C_VEL
LIN {X 0,Y 98.159,Z 593.641,A -85,B 0,C 180,E1 -28589.229,E2 -28589.229} C_VEL
LIN {X 0,Y 107.95,Z 586.097,A -85,B 0,C 180,E1 -28593.536,E2 -28593.536} C_VEL
LIN {X 0,Y 118.314,Z 577.02,A -85,B 0,C 180,E1 -28597.036,E2 -28597.036} C_VEL
LIN {X 0,Y 129.079,Z 566.118,A -85,B 0,C 180,E1 -28599.925,E2 -28599.925} C_VEL
LIN {X 0,Y 139.337,Z 553.865,A -85,B 0,C 180,E1 -28602.187,E2 -28602.187} C_VEL
LIN {X 0,Y 148.141,Z 541.372,A -85,B 0,C 180,E1 -28603.886,E2 -28603.886} C_VEL
LIN {X 0,Y 152.676,Z 533.988,A -85,B 0,C 180,E1 -28604.648,E2 -28604.648} C_VEL
LIN {X 0,Y 155.311,Z 529.054,A -85,B 0,C 180,E1 -28605.32,E2 -28605.32} C_VEL
LIN {X 0,Y 161.374,Z 514.188,A -85,B 0,C 180,E1 -28608.158,E2 -28608.158} C_VEL
LIN {X 0,Y 163.375,Z 508.936,A -85,B 0,C 180,E1 -28608.794,E2 -28608.794} C_VEL
LIN {X 0,Y 164.079,Z 507.131,A -85,B 0,C 180,E1 -28608.912,E2 -28608.912} C_VEL
LIN {X 0,Y 169.311,Z 492.028,A -85,B 0,C 180,E1 -28609.507,E2 -28609.507} C_VEL
LIN {X 0,Y 173.221,Z 476.271,A -85,B 0,C 180,E1 -28609.957,E2 -28609.957} C_VEL
LIN {X 0,Y 175.47,Z 462.374,A -85,B 0,C 180,E1 -28610.214,E2 -28610.214} C_VEL
LIN {X 0,Y 176.932,Z 449.558,A -85,B 0,C 180,E1 -28610.493,E2 -28610.493} C_VEL
LIN {X 0,Y 176.001,Z 446.449,A -85,B 0,C 180,E1 -28613.408,E2 -28613.408} C_VEL
LIN {X 0,Y 175.553,Z 444.96,A -85,B 0,C 180,E1 -28615.408,E2 -28615.408} C_VEL
LIN {X 0,Y 175.244,Z 442.533,A -85,B 0,C 180,E1 -28619.237,E2 -28619.237} C_VEL
LIN {X 0,Y 175.234,Z 442.656,A -85,B 0,C 180,E1 -28621.437,E2 -28621.437} C_VEL
LIN {X 0,Y 175.881,Z 446.165,A -85,B 0,C 180,E1 -28626.741,E2 -28626.741} C_VEL
LIN {X 0,Y 176.834,Z 449.263,A -85,B 0,C 180,E1 -28629.832,E2 -28629.832} C_VEL
LIN {X 0,Y 176.893,Z 449.491,A -85,B 0,C 180,E1 -28630,E2 -28630} C_VEL
LIN {X 0,Y 174.229,Z 469.838,A -85,B 0,C 180,E1 -28630.471,E2 -28630.471} C_VEL
LIN {X 0,Y 171.015,Z 484.518,A -85,B 0,C 180,E1 -28630.905,E2 -28630.905} C_VEL
LIN {X 0,Y 166.707,Z 498.609,A -85,B 0,C 180,E1 -28631.501,E2 -28631.501} C_VEL
LIN {X 0,Y 160.973,Z 512.969,A -85,B 0,C 180,E1 -28632.338,E2 -28632.338} C_VEL
LIN {X 0,Y 153.915,Z 527.065,A -85,B 0,C 180,E1 -28633.484,E2 -28633.484} C_VEL
LIN {X 0,Y 146.314,Z 539.574,A -85,B 0,C 180,E1 -28634.826,E2 -28634.826} C_VEL
LIN {X 0,Y 137.407,Z 551.757,A -85,B 0,C 180,E1 -28636.455,E2 -28636.455} C_VEL
LIN {X 0,Y 127.825,Z 562.855,A -85,B 0,C 180,E1 -28638.476,E2 -28638.476} C_VEL
LIN {X 0,Y 117.312,Z 573.3,A -85,B 0,C 180,E1 -28641.245,E2 -28641.245} C_VEL
LIN {X 0,Y 107.925,Z 581.33,A -85,B 0,C 180,E1 -28644.258,E2 -28644.258} C_VEL
LIN {X 0,Y 99.104,Z 587.944,A -85,B 0,C 180,E1 -28647.566,E2 -28647.566} C_VEL
LIN {X 0,Y 87.984,Z 595.248,A -85,B 0,C 180,E1 -28652.991,E2 -28652.991} C_VEL
LIN {X 0,Y 77.853,Z 601.029,A -85,B 0,C 180,E1 -28659.882,E2 -28659.882} C_VEL
LIN {X 0,Y 71.129,Z 604.445,A -85,B 0,C 180,E1 -28666.236,E2 -28666.236} C_VEL
LIN {X 0,Y 63.623,Z 607.895,A -85,B 0,C 180,E1 -28676.47,E2 -28676.47} C_VEL
LIN {X 0,Y 58.471,Z 610.159,A -85,B 0,C 180,E1 -28688.86,E2 -28688.86} C_VEL
LIN {X 0,Y 56.023,Z 611.298,A -85,B 0,C 180,E1 -28702.79,E2 -28702.79} C_VEL
LIN {X 0,Y 55.808,Z 611.447,A -85,B 0,C 180,E1 -28709.997,E2 -28709.997} C_VEL
LIN {X 0,Y 56.899,Z 610.895,A -85,B 0,C 180,E1 -28724.299,E2 -28724.299} C_VEL
LIN {X 0,Y 60.706,Z 609.237,A -85,B 0,C 180,E1 -28737.583,E2 -28737.583} C_VEL
LIN {X 0,Y 67.023,Z 606.426,A -85,B 0,C 180,E1 -28748.984,E2 -28748.984} C_VEL
LIN {X 0,Y 75.425,Z 602.385,A -85,B 0,C 180,E1 -28758.192,E2 -28758.192} C_VEL
LIN {X 0,Y 85.268,Z 597.018,A -85,B 0,C 180,E1 -28765.507,E2 -28765.507} C_VEL
LIN {X 0,Y 96.19,Z 590.165,A -85,B 0,C 180,E1 -28771.251,E2 -28771.251} C_VEL
LIN {X 0,Y 106.361,Z 582.795,A -85,B 0,C 180,E1 -28775.302,E2 -28775.302} C_VEL
LIN {X 0,Y 115.03,Z 575.546,A -85,B 0,C 180,E1 -28778.172,E2 -28778.172} C_VEL
LIN {X 0,Y 124.632,Z 566.445,A -85,B 0,C 180,E1 -28780.823,E2 -28780.823} C_VEL
LIN {X 0,Y 134.163,Z 556.049,A -85,B 0,C 180,E1 -28782.937,E2 -28782.937} C_VEL
LIN {X 0,Y 142.985,Z 544.74,A -85,B 0,C 180,E1 -28784.707,E2 -28784.707} C_VEL
LIN {X 0,Y 151.122,Z 532.44,A -85,B 0,C 180,E1 -28786.115,E2 -28786.115} C_VEL
LIN {X 0,Y 158.457,Z 518.987,A -85,B 0,C 180,E1 -28787.355,E2 -28787.355} C_VEL
LIN {X 0,Y 164.647,Z 505.024,A -85,B 0,C 180,E1 -28788.259,E2 -28788.259} C_VEL
LIN {X 0,Y 169.621,Z 490.66,A -85,B 0,C 180,E1 -28788.943,E2 -28788.943} C_VEL
LIN {X 0,Y 173.477,Z 475.402,A -85,B 0,C 180,E1 -28789.515,E2 -28789.515} C_VEL
LIN {X 0,Y 176.05,Z 459.695,A -85,B 0,C 180,E1 -28789.87,E2 -28789.87} C_VEL
LIN {X 0,Y 177.18,Z 449.783,A -85,B 0,C 180,E1 -28790.078,E2 -28790.078} C_VEL
LIN {X 0,Y 176.103,Z 446.057,A -85,B 0,C 180,E1 -28793.688,E2 -28793.688} C_VEL
LIN {X 0,Y 175.538,Z 442.655,A -85,B 0,C 180,E1 -28799.426,E2 -28799.426} C_VEL
LIN {X 0,Y 175.532,Z 442.849,A -85,B 0,C 180,E1 -28800.645,E2 -28800.645} C_VEL
LIN {X 0,Y 176.217,Z 446.441,A -85,B 0,C 180,E1 -28806.296,E2 -28806.296} C_VEL
LIN {X 0,Y 177.078,Z 449.367,A -85,B 0,C 180,E1 -28809.134,E2 -28809.134} C_VEL
LIN {X 0,Y 177.213,Z 449.747,A -85,B 0,C 180,E1 -28809.484,E2 -28809.484} C_VEL
LIN {X 0,Y 174.445,Z 471.296,A -85,B 0,C 180,E1 -28809.927,E2 -28809.927} C_VEL
LIN {X 0,Y 171.103,Z 486.619,A -85,B 0,C 180,E1 -28810.306,E2 -28810.306} C_VEL
LIN {X 0,Y 166.799,Z 500.691,A -85,B 0,C 180,E1 -28810.812,E2 -28810.812} C_VEL
LIN {X 0,Y 161.318,Z 514.406,A -85,B 0,C 180,E1 -28811.416,E2 -28811.416} C_VEL
LIN {X 0,Y 154.623,Z 527.849,A -85,B 0,C 180,E1 -28812.256,E2 -28812.256} C_VEL
LIN {X 0,Y 146.322,Z 541.545,A -85,B 0,C 180,E1 -28813.442,E2 -28813.442} C_VEL
LIN {X 0,Y 137.322,Z 553.964,A -85,B 0,C 180,E1 -28814.988,E2 -28814.988} C_VEL
LIN {X 0,Y 126.816,Z 566.14,A -85,B 0,C 180,E1 -28817.069,E2 -28817.069} C_VEL
LIN {X 0,Y 117.283,Z 575.549,A -85,B 0,C 180,E1 -28819.306,E2 -28819.306} C_VEL
LIN {X 0,Y 106.443,Z 584.808,A -85,B 0,C 180,E1 -28822.432,E2 -28822.432} C_VEL
LIN {X 0,Y 94.703,Z 593.549,A -85,B 0,C 180,E1 -28827.064,E2 -28827.064} C_VEL
LIN {X 0,Y 83.664,Z 600.57,A -85,B 0,C 180,E1 -28832.861,E2 -28832.861} C_VEL
LIN {X 0,Y 73.745,Z 606.105,A -85,B 0,C 180,E1 -28840.326,E2 -28840.326} C_VEL
LIN {X 0,Y 65.437,Z 610.307,A -85,B 0,C 180,E1 -28849.883,E2 -28849.883} C_VEL
LIN {X 0,Y 59.252,Z 613.267,A -85,B 0,C 180,E1 -28861.68,E2 -28861.68} C_VEL
LIN {X 0,Y 55.979,Z 615.056,A -85,B 0,C 180,E1 -28875.461,E2 -28875.461} C_VEL
LIN {X 0,Y 55.594,Z 615.691,A -85,B 0,C 180,E1 -28890.003,E2 -28890.003} C_VEL
LIN {X 0,Y 55.98,Z 615.034,A -85,B 0,C 180,E1 -28904.545,E2 -28904.545} C_VEL
LIN {X 0,Y 59.256,Z 613.214,A -85,B 0,C 180,E1 -28918.325,E2 -28918.325} C_VEL
LIN {X 0,Y 65.454,Z 610.229,A -85,B 0,C 180,E1 -28930.112,E2 -28930.112} C_VEL
LIN {X 0,Y 73.745,Z 606.003,A -85,B 0,C 180,E1 -28939.681,E2 -28939.681} C_VEL
LIN {X 0,Y 83.651,Z 600.431,A -85,B 0,C 180,E1 -28947.161,E2 -28947.161} C_VEL
LIN {X 0,Y 94.689,Z 593.366,A -85,B 0,C 180,E1 -28952.961,E2 -28952.961} C_VEL
LIN {X 0,Y 104.948,Z 585.822,A -85,B 0,C 180,E1 -28957.047,E2 -28957.047} C_VEL
LIN {X 0,Y 115.711,Z 576.745,A -85,B 0,C 180,E1 -28960.299,E2 -28960.299} C_VEL
LIN {X 0,Y 125.197,Z 567.487,A -85,B 0,C 180,E1 -28962.618,E2 -28962.618} C_VEL
LIN {X 0,Y 134.879,Z 556.589,A -85,B 0,C 180,E1 -28964.577,E2 -28964.577} C_VEL
LIN {X 0,Y 143.772,Z 544.812,A -85,B 0,C 180,E1 -28966.16,E2 -28966.16} C_VEL
LIN {X 0,Y 152.125,Z 531.69,A -85,B 0,C 180,E1 -28967.416,E2 -28967.416} C_VEL
LIN {X 0,Y 158.788,Z 519.087,A -85,B 0,C 180,E1 -28968.317,E2 -28968.317} C_VEL
LIN {X 0,Y 164.079,Z 507.131,A -85,B 0,C 180,E1 -28968.912,E2 -28968.912} C_VEL
LIN {X 0,Y 166.001,Z 501.701,A -85,B 0,C 180,E1 -28969.374,E2 -28969.374} C_VEL
LIN {X 0,Y 168.425,Z 492.826,A -85,B 0,C 180,E1 -28970.639,E2 -28970.639} C_VEL
LIN {X 0,Y 170.462,Z 483.803,A -85,B 0,C 180,E1 -28971.851,E2 -28971.851} C_VEL
LIN {X 0,Y 171.662,Z 478.139,A -85,B 0,C 180,E1 -28972.24,E2 -28972.24} C_VEL
LIN {X 0,Y 174.261,Z 463.094,A -85,B 0,C 180,E1 -28972.498,E2 -28972.498} C_VEL
LIN {X 0,Y 175.285,Z 454.399,A -85,B 0,C 180,E1 -28972.719,E2 -28972.719} C_VEL
LIN {X 0,Y 174.676,Z 452.126,A -85,B 0,C 180,E1 -28975.385,E2 -28975.385} C_VEL
LIN {X 0,Y 174.365,Z 449.469,A -85,B 0,C 180,E1 -28980,E2 -28980} C_VEL
LIN {X 0,Y 174.348,Z 449.824,A -85,B 0,C 180,E1 -28981.342,E2 -28981.342} C_VEL
LIN {X 0,Y 174.889,Z 453.128,A -85,B 0,C 180,E1 -28986.345,E2 -28986.345} C_VEL
LIN {X 0,Y 175.258,Z 454.49,A -85,B 0,C 180,E1 -28987.824,E2 -28987.824} C_VEL
LIN {X 0,Y 173.067,Z 470.194,A -85,B 0,C 180,E1 -28988.163,E2 -28988.163} C_VEL
LIN {X 0,Y 169.667,Z 485.326,A -85,B 0,C 180,E1 -28988.566,E2 -28988.566} C_VEL
LIN {X 0,Y 164.929,Z 500.255,A -85,B 0,C 180,E1 -28989.162,E2 -28989.162} C_VEL
LIN {X 0,Y 159.607,Z 513.245,A -85,B 0,C 180,E1 -28989.848,E2 -28989.848} C_VEL
LIN {X 0,Y 152.233,Z 527.649,A -85,B 0,C 180,E1 -28990.912,E2 -28990.912} C_VEL
LIN {X 0,Y 144.661,Z 539.848,A -85,B 0,C 180,E1 -28992.11,E2 -28992.11} C_VEL
LIN {X 0,Y 135.567,Z 552.03,A -85,B 0,C 180,E1 -28993.576,E2 -28993.576} C_VEL
LIN {X 0,Y 125.76,Z 563.127,A -85,B 0,C 180,E1 -28995.414,E2 -28995.414} C_VEL
LIN {X 0,Y 115.88,Z 572.678,A -85,B 0,C 180,E1 -28997.653,E2 -28997.653} C_VEL
LIN {X 0,Y 105.211,Z 581.602,A -85,B 0,C 180,E1 -29000.736,E2 -29000.736} C_VEL
LIN {X 0,Y 96.022,Z 588.217,A -85,B 0,C 180,E1 -29003.804,E2 -29003.804} C_VEL
LIN {X 0,Y 84.311,Z 595.521,A -85,B 0,C 180,E1 -29008.92,E2 -29008.92} C_VEL
LIN {X 0,Y 73.491,Z 601.301,A -85,B 0,C 180,E1 -29015.619,E2 -29015.619} C_VEL
LIN {X 0,Y 66.168,Z 604.717,A -85,B 0,C 180,E1 -29021.964,E2 -29021.964} C_VEL
LIN {X 0,Y 57.806,Z 608.168,A -85,B 0,C 180,E1 -29032.558,E2 -29032.558} C_VEL
LIN {X 0,Y 51.903,Z 610.43,A -85,B 0,C 180,E1 -29046.028,E2 -29046.028} C_VEL
LIN {X 0,Y 48.986,Z 611.569,A -85,B 0,C 180,E1 -29061.747,E2 -29061.747} C_VEL
LIN {X 0,Y 48.728,Z 611.717,A -85,B 0,C 180,E1 -29069.996,E2 -29069.996} C_VEL
LIN {X 0,Y 50.053,Z 611.165,A -85,B 0,C 180,E1 -29086.305,E2 -29086.305} C_VEL
LIN {X 0,Y 54.506,Z 609.507,A -85,B 0,C 180,E1 -29101.044,E2 -29101.044} C_VEL
LIN {X 0,Y 61.649,Z 606.697,A -85,B 0,C 180,E1 -29113.153,E2 -29113.153} C_VEL
LIN {X 0,Y 70.866,Z 602.656,A -85,B 0,C 180,E1 -29122.498,E2 -29122.498} C_VEL
LIN {X 0,Y 81.451,Z 597.288,A -85,B 0,C 180,E1 -29129.634,E2 -29129.634} C_VEL
LIN {X 0,Y 92.97,Z 590.435,A -85,B 0,C 180,E1 -29135.107,E2 -29135.107} C_VEL
LIN {X 0,Y 103.597,Z 583.063,A -85,B 0,C 180,E1 -29138.87,E2 -29138.87} C_VEL
LIN {X 0,Y 113.333,Z 575.159,A -85,B 0,C 180,E1 -29141.768,E2 -29141.768} C_VEL
LIN {X 0,Y 124.093,Z 565.097,A -85,B 0,C 180,E1 -29144.316,E2 -29144.316} C_VEL
LIN {X 0,Y 133.883,Z 554.377,A -85,B 0,C 180,E1 -29146.194,E2 -29146.194} C_VEL
LIN {X 0,Y 142.951,Z 542.668,A -85,B 0,C 180,E1 -29147.717,E2 -29147.717} C_VEL
LIN {X 0,Y 151.549,Z 529.342,A -85,B 0,C 180,E1 -29149.06,E2 -29149.06} C_VEL
LIN {X 0,Y 158.726,Z 515.747,A -85,B 0,C 180,E1 -29150.116,E2 -29150.116} C_VEL
LIN {X 0,Y 164.954,Z 501.027,A -85,B 0,C 180,E1 -29150.904,E2 -29150.904} C_VEL
LIN {X 0,Y 169.806,Z 485.975,A -85,B 0,C 180,E1 -29151.494,E2 -29151.494} C_VEL
LIN {X 0,Y 173.19,Z 471.198,A -85,B 0,C 180,E1 -29151.93,E2 -29151.93} C_VEL
LIN {X 0,Y 175.552,Z 454.751,A -85,B 0,C 180,E1 -29152.254,E2 -29152.254} C_VEL
LIN {X 0,Y 174.924,Z 452.324,A -85,B 0,C 180,E1 -29155.102,E2 -29155.102} C_VEL
LIN {X 0,Y 174.669,Z 449.727,A -85,B 0,C 180,E1 -29159.423,E2 -29159.423} C_VEL
LIN {X 0,Y 174.655,Z 449.919,A -85,B 0,C 180,E1 -29160.432,E2 -29160.432} C_VEL
LIN {X 0,Y 175.192,Z 453.267,A -85,B 0,C 180,E1 -29165.756,E2 -29165.756} C_VEL
LIN {X 0,Y 175.569,Z 454.654,A -85,B 0,C 180,E1 -29167.269,E2 -29167.269} C_VEL
LIN {X 0,Y 173.098,Z 472.453,A -85,B 0,C 180,E1 -29167.641,E2 -29167.641} C_VEL
LIN {X 0,Y 169.349,Z 488.584,A -85,B 0,C 180,E1 -29168,E2 -29168} C_VEL
LIN {X 0,Y 164.306,Z 503.899,A -85,B 0,C 180,E1 -29168.526,E2 -29168.526} C_VEL
LIN {X 0,Y 158.361,Z 517.698,A -85,B 0,C 180,E1 -29169.095,E2 -29169.095} C_VEL
LIN {X 0,Y 151.579,Z 530.503,A -85,B 0,C 180,E1 -29169.856,E2 -29169.856} C_VEL
LIN {X 0,Y 143.155,Z 543.657,A -85,B 0,C 180,E1 -29170.932,E2 -29170.932} C_VEL
LIN {X 0,Y 134.22,Z 555.414,A -85,B 0,C 180,E1 -29172.309,E2 -29172.309} C_VEL
LIN {X 0,Y 124.905,Z 565.871,A -85,B 0,C 180,E1 -29173.934,E2 -29173.934} C_VEL
LIN {X 0,Y 115.109,Z 575.277,A -85,B 0,C 180,E1 -29175.931,E2 -29175.931} C_VEL
LIN {X 0,Y 103.92,Z 584.537,A -85,B 0,C 180,E1 -29178.778,E2 -29178.778} C_VEL
LIN {X 0,Y 91.668,Z 593.278,A -85,B 0,C 180,E1 -29183.077,E2 -29183.077} C_VEL
LIN {X 0,Y 79.999,Z 600.298,A -85,B 0,C 180,E1 -29188.541,E2 -29188.541} C_VEL
LIN {X 0,Y 69.311,Z 605.832,A -85,B 0,C 180,E1 -29195.792,E2 -29195.792} C_VEL
LIN {X 0,Y 60.128,Z 610.034,A -85,B 0,C 180,E1 -29205.472,E2 -29205.472} C_VEL
LIN {X 0,Y 53.062,Z 612.995,A -85,B 0,C 180,E1 -29218.013,E2 -29218.013} C_VEL
LIN {X 0,Y 49.079,Z 614.784,A -85,B 0,C 180,E1 -29233.362,E2 -29233.362} C_VEL
LIN {X 0,Y 48.48,Z 615.42,A -85,B 0,C 180,E1 -29250.004,E2 -29250.004} C_VEL
LIN {X 0,Y 49.08,Z 614.761,A -85,B 0,C 180,E1 -29266.646,E2 -29266.646} C_VEL
LIN {X 0,Y 53.067,Z 612.941,A -85,B 0,C 180,E1 -29281.993,E2 -29281.993} C_VEL
LIN {X 0,Y 60.143,Z 609.955,A -85,B 0,C 180,E1 -29294.523,E2 -29294.523} C_VEL
LIN {X 0,Y 69.311,Z 605.728,A -85,B 0,C 180,E1 -29304.217,E2 -29304.217} C_VEL
LIN {X 0,Y 79.99,Z 600.156,A -85,B 0,C 180,E1 -29311.48,E2 -29311.48} C_VEL
LIN {X 0,Y 91.648,Z 593.091,A -85,B 0,C 180,E1 -29316.964,E2 -29316.964} C_VEL
LIN {X 0,Y 102.359,Z 585.546,A -85,B 0,C 180,E1 -29320.754,E2 -29320.754} C_VEL
LIN {X 0,Y 113.497,Z 576.47,A -85,B 0,C 180,E1 -29323.704,E2 -29323.704} C_VEL
LIN {X 0,Y 124.901,Z 565.569,A -85,B 0,C 180,E1 -29326.087,E2 -29326.087} C_VEL
LIN {X 0,Y 135.232,Z 553.848,A -85,B 0,C 180,E1 -29327.879,E2 -29327.879} C_VEL
LIN {X 0,Y 144.839,Z 540.823,A -85,B 0,C 180,E1 -29329.3,E2 -29329.3} C_VEL
LIN {X 0,Y 152.424,Z 528.551,A -85,B 0,C 180,E1 -29330.26,E2 -29330.26} C_VEL
LIN {X 0,Y 159.21,Z 515.273,A -85,B 0,C 180,E1 -29331.013,E2 -29331.013} C_VEL
LIN {X 0,Y 165.056,Z 501.076,A -85,B 0,C 180,E1 -29331.572,E2 -29331.572} C_VEL
LIN {X 0,Y 169.785,Z 485.939,A -85,B 0,C 180,E1 -29332.046,E2 -29332.046} C_VEL
LIN {X 0,Y 171.662,Z 478.139,A -85,B 0,C 180,E1 -29332.24,E2 -29332.24} C_VEL
LIN {X 0,Y 172.366,Z 474.533,A -85,B 0,C 180,E1 -29332.495,E2 -29332.495} C_VEL
LIN {X 0,Y 173.007,Z 469.481,A -85,B 0,C 180,E1 -29333.315,E2 -29333.315} C_VEL
LIN {X 0,Y 173.306,Z 465.058,A -85,B 0,C 180,E1 -29334.505,E2 -29334.505} C_VEL
LIN {X 0,Y 173.415,Z 461.307,A -85,B 0,C 180,E1 -29335.986,E2 -29335.986} C_VEL
LIN {X 0,Y 173.447,Z 458.46,A -85,B 0,C 180,E1 -29337.668,E2 -29337.668} C_VEL
LIN {X 0,Y 173.467,Z 457.186,A -85,B 0,C 180,E1 -29338.881,E2 -29338.881} C_VEL
LIN {X 0,Y 173.497,Z 456.539,A -85,B 0,C 180,E1 -29340,E2 -29340} C_VEL
LIN {X 0,Y 173.461,Z 457.054,A -85,B 0,C 180,E1 -29341.349,E2 -29341.349} C_VEL
LIN {X 0,Y 173.839,Z 459.747,A -85,B 0,C 180,E1 -29345.576,E2 -29345.576} C_VEL
LIN {X 0,Y 171.988,Z 471.625,A -85,B 0,C 180,E1 -29345.849,E2 -29345.849} C_VEL
LIN {X 0,Y 168.312,Z 487.19,A -85,B 0,C 180,E1 -29346.235,E2 -29346.235} C_VEL
LIN {X 0,Y 163.496,Z 501.732,A -85,B 0,C 180,E1 -29346.768,E2 -29346.768} C_VEL
LIN {X 0,Y 157.704,Z 515.278,A -85,B 0,C 180,E1 -29347.439,E2 -29347.439} C_VEL
LIN {X 0,Y 150.887,Z 528.197,A -85,B 0,C 180,E1 -29348.285,E2 -29348.285} C_VEL
LIN {X 0,Y 142.491,Z 541.291,A -85,B 0,C 180,E1 -29349.434,E2 -29349.434} C_VEL
LIN {X 0,Y 134.076,Z 552.304,A -85,B 0,C 180,E1 -29350.621,E2 -29350.621} C_VEL
LIN {X 0,Y 124.059,Z 563.401,A -85,B 0,C 180,E1 -29352.244,E2 -29352.244} C_VEL
LIN {X 0,Y 113.453,Z 573.378,A -85,B 0,C 180,E1 -29354.347,E2 -29354.347} C_VEL
LIN {X 0,Y 102.914,Z 581.874,A -85,B 0,C 180,E1 -29357.041,E2 -29357.041} C_VEL
LIN {X 0,Y 93.379,Z 588.489,A -85,B 0,C 180,E1 -29359.81,E2 -29359.81} C_VEL
LIN {X 0,Y 81.106,Z 595.793,A -85,B 0,C 180,E1 -29364.509,E2 -29364.509} C_VEL
LIN {X 0,Y 69.583,Z 601.573,A -85,B 0,C 180,E1 -29370.844,E2 -29370.844} C_VEL
LIN {X 0,Y 61.633,Z 604.989,A -85,B 0,C 180,E1 -29377.036,E2 -29377.036} C_VEL
LIN {X 0,Y 52.319,Z 608.44,A -85,B 0,C 180,E1 -29387.8,E2 -29387.8} C_VEL
LIN {X 0,Y 45.508,Z 610.7,A -85,B 0,C 180,E1 -29402.395,E2 -29402.395} C_VEL
LIN {X 0,Y 41.989,Z 611.839,A -85,B 0,C 180,E1 -29420.36,E2 -29420.36} C_VEL
LIN {X 0,Y 41.634,Z 611.987,A -85,B 0,C 180,E1 -29429.995,E2 -29429.995} C_VEL
LIN {X 0,Y 43.276,Z 611.435,A -85,B 0,C 180,E1 -29448.949,E2 -29448.949} C_VEL
LIN {X 0,Y 48.53,Z 609.779,A -85,B 0,C 180,E1 -29465.395,E2 -29465.395} C_VEL
LIN {X 0,Y 56.666,Z 606.967,A -85,B 0,C 180,E1 -29478.081,E2 -29478.081} C_VEL
LIN {X 0,Y 66.761,Z 602.927,A -85,B 0,C 180,E1 -29487.364,E2 -29487.364} C_VEL
LIN {X 0,Y 78.084,Z 597.558,A -85,B 0,C 180,E1 -29494.159,E2 -29494.159} C_VEL
LIN {X 0,Y 90.205,Z 590.705,A -85,B 0,C 180,E1 -29499.212,E2 -29499.212} C_VEL
LIN {X 0,Y 101.254,Z 583.332,A -85,B 0,C 180,E1 -29502.621,E2 -29502.621} C_VEL
LIN {X 0,Y 112.214,Z 574.673,A -85,B 0,C 180,E1 -29505.491,E2 -29505.491} C_VEL
LIN {X 0,Y 122.366,Z 565.365,A -85,B 0,C 180,E1 -29507.516,E2 -29507.516} C_VEL
LIN {X 0,Y 132.371,Z 554.644,A -85,B 0,C 180,E1 -29509.175,E2 -29509.175} C_VEL
LIN {X 0,Y 141.611,Z 542.934,A -85,B 0,C 180,E1 -29510.523,E2 -29510.523} C_VEL
LIN {X 0,Y 150.199,Z 529.88,A -85,B 0,C 180,E1 -29511.701,E2 -29511.701} C_VEL
LIN {X 0,Y 157.666,Z 516.011,A -85,B 0,C 180,E1 -29512.648,E2 -29512.648} C_VEL
LIN {X 0,Y 163.507,Z 502.546,A -85,B 0,C 180,E1 -29513.298,E2 -29513.298} C_VEL
LIN {X 0,Y 168.604,Z 487.304,A -85,B 0,C 180,E1 -29513.834,E2 -29513.834} C_VEL
LIN {X 0,Y 172.121,Z 472.609,A -85,B 0,C 180,E1 -29514.238,E2 -29514.238} C_VEL
LIN {X 0,Y 174.13,Z 460.009,A -85,B 0,C 180,E1 -29514.514,E2 -29514.514} C_VEL
LIN {X 0,Y 173.786,Z 456.918,A -85,B 0,C 180,E1 -29519.42,E2 -29519.42} C_VEL
LIN {X 0,Y 173.774,Z 457.061,A -85,B 0,C 180,E1 -29520.289,E2 -29520.289} C_VEL
LIN {X 0,Y 174.159,Z 459.985,A -85,B 0,C 180,E1 -29525.081,E2 -29525.081} C_VEL
LIN {X 0,Y 171.562,Z 476.089,A -85,B 0,C 180,E1 -29525.361,E2 -29525.361} C_VEL
LIN {X 0,Y 167.484,Z 491.924,A -85,B 0,C 180,E1 -29525.702,E2 -29525.702} C_VEL
LIN {X 0,Y 162.135,Z 506.915,A -85,B 0,C 180,E1 -29526.15,E2 -29526.15} C_VEL
LIN {X 0,Y 155.673,Z 520.96,A -85,B 0,C 180,E1 -29526.688,E2 -29526.688} C_VEL
LIN {X 0,Y 147.953,Z 534.518,A -85,B 0,C 180,E1 -29527.441,E2 -29527.441} C_VEL
LIN {X 0,Y 138.575,Z 548.056,A -85,B 0,C 180,E1 -29528.527,E2 -29528.527} C_VEL
LIN {X 0,Y 128.428,Z 560.257,A -85,B 0,C 180,E1 -29529.939,E2 -29529.939} C_VEL
LIN {X 0,Y 118.349,Z 570.507,A -85,B 0,C 180,E1 -29531.534,E2 -29531.534} C_VEL
LIN {X 0,Y 106.758,Z 580.529,A -85,B 0,C 180,E1 -29533.836,E2 -29533.836} C_VEL
LIN {X 0,Y 95.413,Z 588.867,A -85,B 0,C 180,E1 -29536.758,E2 -29536.758} C_VEL
LIN {X 0,Y 82.889,Z 596.714,A -85,B 0,C 180,E1 -29541.152,E2 -29541.152} C_VEL
LIN {X 0,Y 70.98,Z 602.968,A -85,B 0,C 180,E1 -29546.99,E2 -29546.99} C_VEL
LIN {X 0,Y 60.097,Z 607.82,A -85,B 0,C 180,E1 -29555.06,E2 -29555.06} C_VEL
LIN {X 0,Y 50.853,Z 611.392,A -85,B 0,C 180,E1 -29566.295,E2 -29566.295} C_VEL
LIN {X 0,Y 44.212,Z 613.76,A -85,B 0,C 180,E1 -29581.523,E2 -29581.523} C_VEL
LIN {X 0,Y 41.342,Z 614.976,A -85,B 0,C 180,E1 -29600.217,E2 -29600.217} C_VEL
LIN {X 0,Y 41.386,Z 615.15,A -85,B 0,C 180,E1 -29610.005,E2 -29610.005} C_VEL
LIN {X 0,Y 42.278,Z 614.488,A -85,B 0,C 180,E1 -29629.424,E2 -29629.424} C_VEL
LIN {X 0,Y 47.154,Z 612.669,A -85,B 0,C 180,E1 -29646.601,E2 -29646.601} C_VEL
LIN {X 0,Y 55.243,Z 609.68,A -85,B 0,C 180,E1 -29659.764,E2 -29659.764} C_VEL
LIN {X 0,Y 65.377,Z 605.453,A -85,B 0,C 180,E1 -29669.323,E2 -29669.323} C_VEL
LIN {X 0,Y 76.83,Z 599.882,A -85,B 0,C 180,E1 -29676.176,E2 -29676.176} C_VEL
LIN {X 0,Y 89.073,Z 592.814,A -85,B 0,C 180,E1 -29681.238,E2 -29681.238} C_VEL
LIN {X 0,Y 101.851,Z 584.04,A -85,B 0,C 180,E1 -29685.034,E2 -29685.034} C_VEL
LIN {X 0,Y 113.345,Z 574.735,A -85,B 0,C 180,E1 -29687.585,E2 -29687.585} C_VEL
LIN {X 0,Y 123.383,Z 565.295,A -85,B 0,C 180,E1 -29689.298,E2 -29689.298} C_VEL
LIN {X 0,Y 133.915,Z 553.573,A -85,B 0,C 180,E1 -29690.866,E2 -29690.866} C_VEL
LIN {X 0,Y 142.831,Z 541.788,A -85,B 0,C 180,E1 -29692.003,E2 -29692.003} C_VEL
LIN {X 0,Y 151.383,Z 528.275,A -85,B 0,C 180,E1 -29692.916,E2 -29692.916} C_VEL
LIN {X 0,Y 158.256,Z 514.997,A -85,B 0,C 180,E1 -29693.553,E2 -29693.553} C_VEL
LIN {X 0,Y 164,Z 501.231,A -85,B 0,C 180,E1 -29694.012,E2 -29694.012} C_VEL
LIN {X 0,Y 168.844,Z 486.039,A -85,B 0,C 180,E1 -29694.417,E2 -29694.417} C_VEL
LIN {X 0,Y 172.064,Z 471.752,A -85,B 0,C 180,E1 -29694.694,E2 -29694.694} C_VEL
LIN {X 0,Y 173.865,Z 459.696,A -85,B 0,C 180,E1 -29694.938,E2 -29694.938} C_VEL
LIN {X 0,Y 173.467,Z 457.186,A -85,B 0,C 180,E1 -29698.881,E2 -29698.881} C_VEL
LIN {X 0,Y 173.426,Z 457.188,A -85,B 0,C 180,E1 -29699.755,E2 -29699.755} C_VEL
LIN {X 0,Y 173.262,Z 458.537,A -85,B 0,C 180,E1 -29700.787,E2 -29700.787} C_VEL
LIN {X 0,Y 173.012,Z 460.81,A -85,B 0,C 180,E1 -29701.679,E2 -29701.679} C_VEL
LIN {X 0,Y 172.41,Z 465.825,A -85,B 0,C 180,E1 -29702.808,E2 -29702.808} C_VEL
LIN {X 0,Y 171.734,Z 470.144,A -85,B 0,C 180,E1 -29703.345,E2 -29703.345} C_VEL
LIN {X 0,Y 171.172,Z 473.16,A -85,B 0,C 180,E1 -29703.505,E2 -29703.505} C_VEL
LIN {X 0,Y 167.478,Z 488.22,A -85,B 0,C 180,E1 -29703.853,E2 -29703.853} C_VEL
LIN {X 0,Y 162.735,Z 502.215,A -85,B 0,C 180,E1 -29704.304,E2 -29704.304} C_VEL
LIN {X 0,Y 156.943,Z 515.554,A -85,B 0,C 180,E1 -29704.869,E2 -29704.869} C_VEL
LIN {X 0,Y 149.689,Z 529.034,A -85,B 0,C 180,E1 -29705.642,E2 -29705.642} C_VEL
LIN {X 0,Y 141.501,Z 541.565,A -85,B 0,C 180,E1 -29706.6,E2 -29706.6} C_VEL
LIN {X 0,Y 132.952,Z 552.578,A -85,B 0,C 180,E1 -29707.618,E2 -29707.618} C_VEL
LIN {X 0,Y 122.75,Z 563.674,A -85,B 0,C 180,E1 -29709.007,E2 -29709.007} C_VEL
LIN {X 0,Y 111.422,Z 574.067,A -85,B 0,C 180,E1 -29710.908,E2 -29710.908} C_VEL
LIN {X 0,Y 99.399,Z 583.36,A -85,B 0,C 180,E1 -29713.534,E2 -29713.534} C_VEL
LIN {X 0,Y 87.972,Z 590.758,A -85,B 0,C 180,E1 -29716.522,E2 -29716.522} C_VEL
LIN {X 0,Y 75.294,Z 597.661,A -85,B 0,C 180,E1 -29721.02,E2 -29721.02} C_VEL
LIN {X 0,Y 63.267,Z 603.069,A -85,B 0,C 180,E1 -29727.285,E2 -29727.285} C_VEL
LIN {X 0,Y 52.222,Z 607.141,A -85,B 0,C 180,E1 -29736.143,E2 -29736.143} C_VEL
LIN {X 0,Y 42.948,Z 609.985,A -85,B 0,C 180,E1 -29749.108,E2 -29749.108} C_VEL
LIN {X 0,Y 36.625,Z 611.679,A -85,B 0,C 180,E1 -29767.426,E2 -29767.426} C_VEL
LIN {X 0,Y 34.561,Z 612.256,A -85,B 0,C 180,E1 -29789.994,E2 -29789.994} C_VEL
LIN {X 0,Y 36.621,Z 611.706,A -85,B 0,C 180,E1 -29812.565,E2 -29812.565} C_VEL
LIN {X 0,Y 42.911,Z 610.05,A -85,B 0,C 180,E1 -29830.923,E2 -29830.923} C_VEL
LIN {X 0,Y 52.183,Z 607.238,A -85,B 0,C 180,E1 -29843.902,E2 -29843.902} C_VEL
LIN {X 0,Y 63.202,Z 603.198,A -85,B 0,C 180,E1 -29852.816,E2 -29852.816} C_VEL
LIN {X 0,Y 75.253,Z 597.828,A -85,B 0,C 180,E1 -29859.048,E2 -29859.048} C_VEL
LIN {X 0,Y 87.932,Z 590.974,A -85,B 0,C 180,E1 -29863.551,E2 -29863.551} C_VEL
LIN {X 0,Y 99.364,Z 583.601,A -85,B 0,C 180,E1 -29866.532,E2 -29866.532} C_VEL
LIN {X 0,Y 110.145,Z 575.344,A -85,B 0,C 180,E1 -29868.964,E2 -29868.964} C_VEL
LIN {X 0,Y 121.028,Z 565.633,A -85,B 0,C 180,E1 -29870.804,E2 -29870.804} C_VEL
LIN {X 0,Y 131.223,Z 554.911,A -85,B 0,C 180,E1 -29872.218,E2 -29872.218} C_VEL
LIN {X 0,Y 140.617,Z 543.201,A -85,B 0,C 180,E1 -29873.375,E2 -29873.375} C_VEL
LIN {X 0,Y 149.196,Z 530.382,A -85,B 0,C 180,E1 -29874.386,E2 -29874.386} C_VEL
LIN {X 0,Y 156.052,Z 518.036,A -85,B 0,C 180,E1 -29875.141,E2 -29875.141} C_VEL
LIN {X 0,Y 162.096,Z 504.729,A -85,B 0,C 180,E1 -29875.708,E2 -29875.708} C_VEL
LIN {X 0,Y 167.352,Z 489.809,A -85,B 0,C 180,E1 -29876.178,E2 -29876.178} C_VEL
LIN {X 0,Y 171.185,Z 474.801,A -85,B 0,C 180,E1 -29876.564,E2 -29876.564} C_VEL
LIN {X 0,Y 172.812,Z 465.704,A -85,B 0,C 180,E1 -29876.772,E2 -29876.772} C_VEL
LIN {X 0,Y 172.818,Z 464.13,A -85,B 0,C 180,E1 -29879.417,E2 -29879.417} C_VEL
LIN {X 0,Y 172.808,Z 464.242,A -85,B 0,C 180,E1 -29880.291,E2 -29880.291} C_VEL
LIN {X 0,Y 172.841,Z 465.703,A -85,B 0,C 180,E1 -29882.818,E2 -29882.818} C_VEL
LIN {X 0,Y 169.782,Z 481.236,A -85,B 0,C 180,E1 -29883.08,E2 -29883.08} C_VEL
LIN {X 0,Y 165.661,Z 495.467,A -85,B 0,C 180,E1 -29883.36,E2 -29883.36} C_VEL
LIN {X 0,Y 160.222,Z 509.642,A -85,B 0,C 180,E1 -29883.723,E2 -29883.723} C_VEL
LIN {X 0,Y 153.271,Z 523.881,A -85,B 0,C 180,E1 -29884.215,E2 -29884.215} C_VEL
LIN {X 0,Y 145.471,Z 536.862,A -85,B 0,C 180,E1 -29884.854,E2 -29884.854} C_VEL
LIN {X 0,Y 135.977,Z 549.936,A -85,B 0,C 180,E1 -29885.778,E2 -29885.778} C_VEL
LIN {X 0,Y 125.676,Z 561.78,A -85,B 0,C 180,E1 -29886.983,E2 -29886.983} C_VEL
LIN {X 0,Y 115.425,Z 571.748,A -85,B 0,C 180,E1 -29888.349,E2 -29888.349} C_VEL
LIN {X 0,Y 103.591,Z 581.514,A -85,B 0,C 180,E1 -29890.356,E2 -29890.356} C_VEL
LIN {X 0,Y 93.592,Z 588.594,A -85,B 0,C 180,E1 -29892.535,E2 -29892.535} C_VEL
LIN {X 0,Y 80.573,Z 596.442,A -85,B 0,C 180,E1 -29896.375,E2 -29896.375} C_VEL
LIN {X 0,Y 68.022,Z 602.696,A -85,B 0,C 180,E1 -29901.591,E2 -29901.591} C_VEL
LIN {X 0,Y 56.283,Z 607.548,A -85,B 0,C 180,E1 -29909.07,E2 -29909.07} C_VEL
LIN {X 0,Y 45.933,Z 611.119,A -85,B 0,C 180,E1 -29920.097,E2 -29920.097} C_VEL
LIN {X 0,Y 38.062,Z 613.487,A -85,B 0,C 180,E1 -29936.369,E2 -29936.369} C_VEL
LIN {X 0,Y 34.331,Z 614.704,A -85,B 0,C 180,E1 -29958.193,E2 -29958.193} C_VEL
LIN {X 0,Y 34.276,Z 614.879,A -85,B 0,C 180,E1 -29970.006,E2 -29970.006} C_VEL
LIN {X 0,Y 35.621,Z 614.216,A -85,B 0,C 180,E1 -29993.247,E2 -29993.247} C_VEL
LIN {X 0,Y 41.612,Z 612.395,A -85,B 0,C 180,E1 -30012.505,E2 -30012.505} C_VEL
LIN {X 0,Y 52.592,Z 608.813,A -85,B 0,C 180,E1 -30027.689,E2 -30027.689} C_VEL
LIN {X 0,Y 64.987,Z 603.915,A -85,B 0,C 180,E1 -30036.822,E2 -30036.822} C_VEL
LIN {X 0,Y 77.389,Z 597.973,A -85,B 0,C 180,E1 -30042.476,E2 -30042.476} C_VEL
LIN {X 0,Y 90.323,Z 590.488,A -85,B 0,C 180,E1 -30046.636,E2 -30046.636} C_VEL
LIN {X 0,Y 101.917,Z 582.526,A -85,B 0,C 180,E1 -30049.324,E2 -30049.324} C_VEL
LIN {X 0,Y 113.722,Z 572.965,A -85,B 0,C 180,E1 -30051.428,E2 -30051.428} C_VEL
LIN {X 0,Y 123.972,Z 563.24,A -85,B 0,C 180,E1 -30052.798,E2 -30052.798} C_VEL
LIN {X 0,Y 134.258,Z 551.689,A -85,B 0,C 180,E1 -30054.055,E2 -30054.055} C_VEL
LIN {X 0,Y 142.878,Z 540.27,A -85,B 0,C 180,E1 -30054.938,E2 -30054.938} C_VEL
LIN {X 0,Y 151.536,Z 526.449,A -85,B 0,C 180,E1 -30055.68,E2 -30055.68} C_VEL
LIN {X 0,Y 158.487,Z 512.864,A -85,B 0,C 180,E1 -30056.177,E2 -30056.177} C_VEL
LIN {X 0,Y 164.509,Z 497.952,A -85,B 0,C 180,E1 -30056.577,E2 -30056.577} C_VEL
LIN {X 0,Y 168.926,Z 483.479,A -85,B 0,C 180,E1 -30056.879,E2 -30056.879} C_VEL
LIN {X 0,Y 172.167,Z 468.18,A -85,B 0,C 180,E1 -30057.08,E2 -30057.08} C_VEL
LIN {X 0,Y 172.554,Z 465.38,A -85,B 0,C 180,E1 -30057.218,E2 -30057.218} C_VEL
LIN {X 0,Y 172.555,Z 463.635,A -85,B 0,C 180,E1 -30060,E2 -30060} C_VEL
LIN {X 0,Y 172.5,Z 464.12,A -85,B 0,C 180,E1 -30061.168,E2 -30061.168} C_VEL
LIN {X 0,Y 172.532,Z 465.435,A -85,B 0,C 180,E1 -30063.377,E2 -30063.377} C_VEL
LIN {X 0,Y 171.172,Z 473.16,A -85,B 0,C 180,E1 -30063.505,E2 -30063.505} C_VEL
LIN {X 0,Y 169.924,Z 478.931,A -85,B 0,C 180,E1 -30063.411,E2 -30063.411} C_VEL
LIN {X 0,Y 167.341,Z 488.247,A -85,B 0,C 180,E1 -30062.644,E2 -30062.644} C_VEL
LIN {X 0,Y 164.271,Z 497.452,A -85,B 0,C 180,E1 -30061.882,E2 -30061.882} C_VEL
LIN {X 0,Y 162.188,Z 502.927,A -85,B 0,C 180,E1 -30061.82,E2 -30061.82} C_VEL
LIN {X 0,Y 155.63,Z 517.588,A -85,B 0,C 180,E1 -30062.357,E2 -30062.357} C_VEL
LIN {X 0,Y 149.001,Z 529.567,A -85,B 0,C 180,E1 -30062.942,E2 -30062.942} C_VEL
LIN {X 0,Y 140.863,Z 541.839,A -85,B 0,C 180,E1 -30063.734,E2 -30063.734} C_VEL
LIN {X 0,Y 132.198,Z 552.851,A -85,B 0,C 180,E1 -30064.567,E2 -30064.567} C_VEL
LIN {X 0,Y 121.841,Z 563.947,A -85,B 0,C 180,E1 -30065.71,E2 -30065.71} C_VEL
LIN {X 0,Y 109.814,Z 574.729,A -85,B 0,C 180,E1 -30067.354,E2 -30067.354} C_VEL
LIN {X 0,Y 97.983,Z 583.632,A -85,B 0,C 180,E1 -30069.501,E2 -30069.501} C_VEL
LIN {X 0,Y 86.219,Z 591.03,A -85,B 0,C 180,E1 -30071.985,E2 -30071.985} C_VEL
LIN {X 0,Y 73.042,Z 597.933,A -85,B 0,C 180,E1 -30075.796,E2 -30075.796} C_VEL
LIN {X 0,Y 60.333,Z 603.342,A -85,B 0,C 180,E1 -30081.259,E2 -30081.259} C_VEL
LIN {X 0,Y 48.37,Z 607.413,A -85,B 0,C 180,E1 -30089.326,E2 -30089.326} C_VEL
LIN {X 0,Y 37.846,Z 610.257,A -85,B 0,C 180,E1 -30102.021,E2 -30102.021} C_VEL
LIN {X 0,Y 30.191,Z 611.95,A -85,B 0,C 180,E1 -30122.246,E2 -30122.246} C_VEL
LIN {X 0,Y 27.476,Z 612.526,A -85,B 0,C 180,E1 -30149.993,E2 -30149.993} C_VEL
LIN {X 0,Y 30.186,Z 611.977,A -85,B 0,C 180,E1 -30177.745,E2 -30177.745} C_VEL
LIN {X 0,Y 37.814,Z 610.321,A -85,B 0,C 180,E1 -30198.017,E2 -30198.017} C_VEL
LIN {X 0,Y 48.337,Z 607.508,A -85,B 0,C 180,E1 -30210.728,E2 -30210.728} C_VEL
LIN {X 0,Y 60.279,Z 603.469,A -85,B 0,C 180,E1 -30218.857,E2 -30218.857} C_VEL
LIN {X 0,Y 73.013,Z 598.098,A -85,B 0,C 180,E1 -30224.264,E2 -30224.264} C_VEL
LIN {X 0,Y 86.187,Z 591.244,A -85,B 0,C 180,E1 -30228.095,E2 -30228.095} C_VEL
LIN {X 0,Y 97.954,Z 583.87,A -85,B 0,C 180,E1 -30230.576,E2 -30230.576} C_VEL
LIN {X 0,Y 109.735,Z 575.042,A -85,B 0,C 180,E1 -30232.735,E2 -30232.735} C_VEL
LIN {X 0,Y 120.098,Z 565.901,A -85,B 0,C 180,E1 -30234.15,E2 -30234.15} C_VEL
LIN {X 0,Y 130.452,Z 555.178,A -85,B 0,C 180,E1 -30235.311,E2 -30235.311} C_VEL
LIN {X 0,Y 139.977,Z 543.467,A -85,B 0,C 180,E1 -30236.259,E2 -30236.259} C_VEL
LIN {X 0,Y 148.67,Z 530.647,A -85,B 0,C 180,E1 -30237.104,E2 -30237.104} C_VEL
LIN {X 0,Y 155.613,Z 518.3,A -85,B 0,C 180,E1 -30237.736,E2 -30237.736} C_VEL
LIN {X 0,Y 161.72,Z 504.991,A -85,B 0,C 180,E1 -30238.208,E2 -30238.208} C_VEL
LIN {X 0,Y 167.089,Z 489.864,A -85,B 0,C 180,E1 -30238.609,E2 -30238.609} C_VEL
LIN {X 0,Y 170.956,Z 474.803,A -85,B 0,C 180,E1 -30238.942,E2 -30238.942} C_VEL
LIN {X 0,Y 171.584,Z 471.526,A -85,B 0,C 180,E1 -30239.051,E2 -30239.051} C_VEL
LIN {X 0,Y 171.642,Z 471.206,A -85,B 0,C 180,E1 -30240,E2 -30240} C_VEL
LIN {X 0,Y 171.602,Z 471.504,A -85,B 0,C 180,E1 -30240.52,E2 -30240.52} C_VEL
LIN {X 0,Y 168.235,Z 485.998,A -85,B 0,C 180,E1 -30240.755,E2 -30240.755} C_VEL
LIN {X 0,Y 163.424,Z 500.769,A -85,B 0,C 180,E1 -30241.025,E2 -30241.025} C_VEL
LIN {X 0,Y 157.29,Z 515.133,A -85,B 0,C 180,E1 -30241.315,E2 -30241.315} C_VEL
LIN {X 0,Y 150.287,Z 528.273,A -85,B 0,C 180,E1 -30241.698,E2 -30241.698} C_VEL
LIN {X 0,Y 141.548,Z 541.676,A -85,B 0,C 180,E1 -30242.289,E2 -30242.289} C_VEL
LIN {X 0,Y 132.1,Z 553.737,A -85,B 0,C 180,E1 -30243.049,E2 -30243.049} C_VEL
LIN {X 0,Y 121.542,Z 565.064,A -85,B 0,C 180,E1 -30244.105,E2 -30244.105} C_VEL
LIN {X 0,Y 109.427,Z 575.901,A -85,B 0,C 180,E1 -30245.458,E2 -30245.458} C_VEL
LIN {X 0,Y 97.405,Z 584.94,A -85,B 0,C 180,E1 -30247.226,E2 -30247.226} C_VEL
LIN {X 0,Y 85.544,Z 592.46,A -85,B 0,C 180,E1 -30249.652,E2 -30249.652} C_VEL
LIN {X 0,Y 72.241,Z 599.483,A -85,B 0,C 180,E1 -30253.392,E2 -30253.392} C_VEL
LIN {X 0,Y 59.347,Z 605.015,A -85,B 0,C 180,E1 -30258.679,E2 -30258.679} C_VEL
LIN {X 0,Y 47.239,Z 609.215,A -85,B 0,C 180,E1 -30266.8,E2 -30266.8} C_VEL
LIN {X 0,Y 36.64,Z 612.177,A -85,B 0,C 180,E1 -30279.901,E2 -30279.901} C_VEL
LIN {X 0,Y 29.164,Z 613.966,A -85,B 0,C 180,E1 -30301.194,E2 -30301.194} C_VEL
LIN {X 0,Y 27.148,Z 614.607,A -85,B 0,C 180,E1 -30330.007,E2 -30330.007} C_VEL
LIN {X 0,Y 29.167,Z 613.942,A -85,B 0,C 180,E1 -30358.818,E2 -30358.818} C_VEL
LIN {X 0,Y 36.648,Z 612.121,A -85,B 0,C 180,E1 -30380.102,E2 -30380.102} C_VEL
LIN {X 0,Y 48.406,Z 608.767,A -85,B 0,C 180,E1 -30394.18,E2 -30394.18} C_VEL
LIN {X 0,Y 59.349,Z 604.904,A -85,B 0,C 180,E1 -30401.336,E2 -30401.336} C_VEL
LIN {X 0,Y 72.243,Z 599.334,A -85,B 0,C 180,E1 -30406.625,E2 -30406.625} C_VEL
LIN {X 0,Y 85.537,Z 592.263,A -85,B 0,C 180,E1 -30410.403,E2 -30410.403} C_VEL
LIN {X 0,Y 99.123,Z 583.491,A -85,B 0,C 180,E1 -30413.054,E2 -30413.054} C_VEL
LIN {X 0,Y 111.152,Z 574.186,A -85,B 0,C 180,E1 -30414.801,E2 -30414.801} C_VEL
LIN {X 0,Y 121.546,Z 564.747,A -85,B 0,C 180,E1 -30415.911,E2 -30415.911} C_VEL
LIN {X 0,Y 132.168,Z 553.299,A -85,B 0,C 180,E1 -30416.952,E2 -30416.952} C_VEL
LIN {X 0,Y 141.553,Z 541.237,A -85,B 0,C 180,E1 -30417.733,E2 -30417.733} C_VEL
LIN {X 0,Y 150.292,Z 527.723,A -85,B 0,C 180,E1 -30418.317,E2 -30418.317} C_VEL
LIN {X 0,Y 157.295,Z 514.444,A -85,B 0,C 180,E1 -30418.706,E2 -30418.706} C_VEL
LIN {X 0,Y 163.316,Z 500.198,A -85,B 0,C 180,E1 -30418.996,E2 -30418.996} C_VEL
LIN {X 0,Y 168.233,Z 484.865,A -85,B 0,C 180,E1 -30419.26,E2 -30419.26} C_VEL
LIN {X 0,Y 171.331,Z 471.192,A -85,B 0,C 180,E1 -30419.474,E2 -30419.474} C_VEL
LIN {X 0,Y 171.383,Z 470.818,A -85,B 0,C 180,E1 -30420,E2 -30420} C_VEL
LIN {X 0,Y 171.307,Z 471.239,A -85,B 0,C 180,E1 -30421.069,E2 -30421.069} C_VEL
LIN {X 0,Y 167.591,Z 486.971,A -85,B 0,C 180,E1 -30421.389,E2 -30421.389} C_VEL
LIN {X 0,Y 162.811,Z 501.321,A -85,B 0,C 180,E1 -30421.773,E2 -30421.773} C_VEL
LIN {X 0,Y 162.188,Z 502.927,A -85,B 0,C 180,E1 -30421.82,E2 -30421.82} C_VEL
LIN {X 0,Y 162.049,Z 503.669,A -85,B 0,C 180,E1 -30421.833,E2 -30421.833} C_VEL
